(* CoDeSys 2.3.9.41 project: VOS_Vorkuta_ASU_3_osmos_2.pro *)
(* Libraries: PID_Regulators.lib 6.11.19 15:29:27, GermesLib_1_3.lib 17.9.20 11:40:29, Util.lib 18.5.10 15:14:28, STANDARD.LIB 4.10.05 11:14:46, IECSFC.LIB 13.4.06 15:51:28, SYSLIBTIME.LIB 6.11.19 15:29:28, ANALYZATION.LIB 5.10.99 09:05:06 *)

(* PLC configuration (modules and I/O channels)
Fast discrete inputs [I_SIMPLE_INPUT] node 0, in %IB0 out %QB0 {ChannellName = Fast discrete inputs; Filtrationtime = 10000}
  DD1_DI_1 AT %IX0.0 [BitInput] Авария насоса Р03.01/01 {ChannellName = Enter name}
  DD1_DI_2 AT %IX0.1 [BitInput] Авария насоса Р03.01/02 {ChannellName = Enter name}
  DD1_DI_3 AT %IX0.2 [BitInput] эк.манометр PIS03.01/01 после насоса Р03.01/01 {ChannellName = Enter name}
  DD1_DI_4 AT %IX0.3 [BitInput] эк.манометр PIS03.01/02 после насоса Р03.01/02 {ChannellName = Enter name}
Discrete inputs [ID130] node 1, in %IB1 out %QB1 {ChannellName = Discrete inputs; Filtrationtime_GeneralINP = 10; PinCount = 12; Visibility = No}
  AT %IB1.0 [ByteInput] 8 discrete inputs {ChannellName = Enter name}
  AT %IB1.1 [ByteInput] 4 discrete inputs {ChannellName = Enter name}
Fast discrete outputs [OWEN_ID570] node 2, in %IB2 out %QB2 {ChannellName = Fast discrete outputs; SafeValueBool = FALSE; SafeValueBool = FALSE; SafeValueBool = FALSE; SafeValueBool = FALSE; Visibility = No}
  AT %QX2.0 [BitOutput] Fast discrete output 1 {ChannellName = Enter name}
  AT %QX2.1 [BitOutput] Fast discrete output 2 {ChannellName = Enter name}
  AT %QX2.2 [BitOutput] Fast discrete output 3 {ChannellName = Enter name}
  AT %QX2.3 [BitOutput] Fast discrete output 4 {ChannellName = Enter name}
Discrete outputs [ID131] node 3, in %IB3 out %QB3 {ChannellName = Discrete outputs; SafeValueByte = 0; Visibility = No}
  AT %QB3.0 [ByteOutput] 8 discrete outputs {ChannellName = Enter name}
  AT %QB3.1 [ByteOutput] 8 discrete outputs {ChannellName = Enter name}
DD1_AI_1 AT %IR4.0 [FloatInputP] резерв {ChannellName = Fast analog input; AIN_TYPE = 0-20 mA; Peak_Filtr = 200; Flt_Ch = Off; TauRC = 10; MinFV = 0; MaxFV = 20}
DD1_AI_2 AT %IR4.1 [FloatInputP] датчик давления РТ03.01/01 {ChannellName = Fast analog input; AIN_TYPE = 0-20 mA; Peak_Filtr = 200; Flt_Ch = Off; TauRC = 10; MinFV = 0; MaxFV = 20}
DD1_AI_3 AT %IR4.2 [FloatInputP] датчик давления РТ03.02/01 {ChannellName = Fast analog input; AIN_TYPE = 0-20 mA; Peak_Filtr = 200; Flt_Ch = Off; TauRC = 10; MinFV = 0; MaxFV = 20}
DD1_AI_4 AT %IR4.3 [FloatInputP] датчик давления РТ03.03/01 {ChannellName = Fast analog input; AIN_TYPE = 0-20 mA; Peak_Filtr = 200; Flt_Ch = Off; TauRC = 10; MinFV = 0; MaxFV = 20}
DD1_AI_5 AT %IR4.4 [FloatInputP] датчик давления РТ03.04/01 {ChannellName = Fast analog input; AIN_TYPE = 0-20 mA; Peak_Filtr = 200; Flt_Ch = Off; TauRC = 10; MinFV = 0; MaxFV = 20}
DD1_AI_6 AT %IR4.5 [FloatInputP] кондуктомер QIT03.01/01 осн.осмос {ChannellName = Fast analog input; AIN_TYPE = 0-20 mA; Peak_Filtr = 200; Flt_Ch = Off; TauRC = 10; MinFV = 0; MaxFV = 20}
DD1_AI_7 AT %IR4.6 [FloatInputP] расходомер FIT03.02/01 осн.осмос {ChannellName = Fast analog input; AIN_TYPE = 0-20 mA; Peak_Filtr = 200; Flt_Ch = Off; TauRC = 10; MinFV = 0; MaxFV = 20}
DD1_AI_8 AT %IR4.7 [FloatInputP] расходомер FIT03.03/01 осн.осмос {ChannellName = Fast analog input; AIN_TYPE = 0-20 mA; Peak_Filtr = 200; Flt_Ch = Off; TauRC = 10; MinFV = 0; MaxFV = 20}
AT %IW4.8 [WordInput] AI read time (10ms) {ChannellName = Enter name}
Analog outputs [ID126] node 5, in %IB5 out %QB5 {ChannellName = Analog outputs}
  DD1_AO_1 AT %QR5.0 [FloatOutputP] производительность осн.доз.насоса Р03.02/01 {ChannellName = Analog output; AOUT_TYPE = 4-20 mA; SafeValueREAL = 0.0}
  DD1_AO_2 AT %QR5.1 [FloatOutputP] производительность рез.доз.насоса Р03.02/02 {ChannellName = Analog output; AOUT_TYPE = 4-20 mA; SafeValueREAL = 0.0}
  DD1_AO_3 AT %QR5.2 [FloatOutputP] резерв {ChannellName = Analog output; AOUT_TYPE = 4-20 mA; SafeValueREAL = 0.0}
  DD1_AO_4 AT %QR5.3 [FloatOutputP] резерв {ChannellName = Analog output; AOUT_TYPE = 4-20 mA; SafeValueREAL = 0.0}
Special input [ID103] node 6, in %IB6 out %QB6 {ChannellName = Special input}
  AT %IX6.0 [BitInput] Special input {ChannellName = Enter name}
Special output [ID104] node 7, in %IB7 out %QB7 {ChannellName = Special output}
  AT %QX7.0 [BitOutput] Special output {ChannellName = Enter name}
AT %QD8.0 [DWordOutput] Last address {ChannellName = Enter name}
AT %QW8.1 [WordOutput] Last error {ChannellName = Enter name}
RS-485-1 [COM1_USART] node 0, in %IB8.0 out %QB8.0 {ChannellName = RS-485-1; CommunicationSpeed = 9600; Parity = NO PARITY CHECK; BitLength = 8 bits; StopLength = One stop bit; InterfaceType = RS485; FrameOriented = RTU; Timeout = 5; Visibility = No}
AT %QB8.1.0 [ComChannel] Command (0xff - Start) {ChannellName = Enter name}
Real input module [ID2007] node 0, in %IB8.1.0 out %QB8.1.0 {ChannellName = float input module; ModbusAddress = 512; Command_read_regs = Read holding Registers  (0x03); Visibility = No}
  PT030102rawValue AT %QD8.1.0.0 [FloatOutput] {ChannellName = Enter name}
Real input module [ID2007] node 1, in %IB8.1.1 out %QB8.1.1 {ChannellName = float input module; ModbusAddress = 514; Command_read_regs = Read holding Registers  (0x03); Visibility = No}
  PT030202rawValue AT %QD8.1.1.0 [FloatOutput] {ChannellName = Enter name}
  PT030302rawValue AT %QD8.1.2.0 [FloatOutput] {ChannellName = Enter name}
Real input module [ID2007] node 3, in %IB8.1.3 out %QB8.1.3 {ChannellName = float input module; ModbusAddress = 518; Command_read_regs = Read holding Registers  (0x03); Visibility = No}
  PT030402rawValue AT %QD8.1.3.0 [FloatOutput] {ChannellName = Enter name}
Real input module [ID2007] node 4, in %IB8.1.4 out %QB8.1.4 {ChannellName = float input module; ModbusAddress = 520; Command_read_regs = Read holding Registers  (0x03); Visibility = No}
  QIT030102rawValue AT %QD8.1.4.0 [FloatOutput] {ChannellName = Enter name}
Real input module [ID2007] node 5, in %IB8.1.5 out %QB8.1.5 {ChannellName = float input module; ModbusAddress = 522; Command_read_regs = Read holding Registers  (0x03); Visibility = No}
  FIT030202rawValue AT %QD8.1.5.0 [FloatOutput] {ChannellName = Enter name}
Real input module [ID2007] node 6, in %IB8.1.6 out %QB8.1.6 {ChannellName = float input module; ModbusAddress = 524; Command_read_regs = Read holding Registers  (0x03); Visibility = No}
  FIT030302rawValue AT %QD8.1.6.0 [FloatOutput] {ChannellName = Enter name}
Real input module [ID2007] node 7, in %IB8.1.7 out %QB8.1.7 {ChannellName = float input module; ModbusAddress = 526; Command_read_regs = Read holding Registers  (0x03); Visibility = No}
  FIT030101rawValue AT %QD8.1.7.0 [FloatOutput] {ChannellName = Enter name}
Register input module [ID2003] node 8, in %IB8.1.8 out %QB8.1.8 {ChannellName = Register input module; ModbusAddress = 529; Command_read_regs = Read input registers  (0x04); Visibility = No}
  DI_bit_mask_DD2 AT %QW8.1.8.0 [WordOutput] {ChannellName = Enter name}
Register input module [ID2003] node 9, in %IB8.1.9 out %QB8.1.9 {ChannellName = Register input module; ModbusAddress = 532; Command_read_regs = Read input registers  (0x04); Visibility = No}
  stat_word_P030601_PLC AT %QW8.1.9.0 [WordOutput] {ChannellName = Enter name}
  stat_word_P030602_PLC AT %QW8.1.10.0 [WordOutput] {ChannellName = Enter name}
Universal Modbus device [ID2000] node 2, in %IB8.2 out %QB8.2 {ChannellName = Universal Modbus device; ModuleIP = 10:0:0:223; ServiceTimeout = 150; TCPport = 502; NetMode = Serial; ModuleSlaveAddress = 1; RequestType = By value change; PeriodOfService = 100; Visibility = No; RepeatCounter = 0; ByteSequence = Native}
  AT %QB8.2.0 [ComChannel] Command (0xff - Start) {ChannellName = Enter name}
  Register output module [ID2004] node 0, in %IB8.2.0 out %QB8.2.0 {ChannellName = Register; ModbusAddress = 528; Command_write_one_reg = Write multiple registers(0x10); Visibility = No}
    DO_bit_mask_DD2 AT %QW8.2.0.0 [WordOutput] {ChannellName = Enter name}
  Register output module [ID2004] node 1, in %IB8.2.1 out %QB8.2.1 {ChannellName = Register; ModbusAddress = 530; Command_write_one_reg = Write multiple registers(0x10); Visibility = No}
    com_word_P030601_PLC AT %QW8.2.1.0 [WordOutput] {ChannellName = Enter name}
  Register output module [ID2004] node 2, in %IB8.2.2 out %QB8.2.2 {ChannellName = Register; ModbusAddress = 531; Command_write_one_reg = Write multiple registers(0x10); Visibility = No}
    set_freq_P030601_PLC AT %QW8.2.2.0 [WordOutput] {ChannellName = Enter name}
  Register output module [ID2004] node 3, in %IB8.2.3 out %QB8.2.3 {ChannellName = Register; ModbusAddress = 533; Command_write_one_reg = Write multiple registers(0x10); Visibility = No}
    com_word_P030602_PLC AT %QW8.2.3.0 [WordOutput] {ChannellName = Enter name}
    set_freq_P030602_PLC AT %QW8.2.4.0 [WordOutput] {ChannellName = Enter name}
RS-232 [COM2_USART] node 0, in %IB9.0.0 out %QB9.0.0 {ChannellName = RS-232; CommunicationSpeed = 115200; Parity = NO PARITY CHECK; BitLength = 8 bits; StopLength = One stop bit; InterfaceType = RS232; FrameOriented = RTU; Timeout = 0; Visibility = No}
*)

(* POU PLC_PRG, CFC *)
PROGRAM PLC_PRG
VAR
	boolStub: BOOL; (*Заглушка bool*)
	realStub: REAL; (*Заглушка real*)
	P0301: RichTwoPumpManager;		(*управление насосами Р03.01 на входе в осмос*)
	resetAlarms: BOOL;		(*Сброс аварий в осмос 2 (МЕ03)*)
	delayCheckIfP030101works: TON;		(*задержка на разгон насоса Р03.01/01*)
	delayCheckIfP030102works: TON;		(*задержка на разгон насоса Р03.01/02*)
	statWordP0301: WORD;		(*статусы состояния насосов Р03.01*)
	lowLevelV0207: BOOL;		(*низкий уровень в емкости V02.07, сигнал из АСУ-2 осмос-1*)
	highLevelV0601: BOOL;		(*высокий уровень в емкости V06.01 сигнал из АСУ-1 общий.*)
	highLevelV0401: BOOL;		(*высокий уровень в емкости V04.01, сигнал из МЕ04, от БМТ.*)
	toNextStarnP030101timer: WORD;		(*Обратный отсчет до возможности повторного пуска насоса Р03.01/01*)
	toNextStarnP030102timer: WORD;		(*обратный отсчет до возможности повторного пуска насоса Р03.01/02*)
	flowFIT0301: REAL;		(*Показания расходомера FIT03.01/01 на входе в осмос 2.
			Для управления производительностью НД Р03.02 (1 и 2).*)
	P0302: RichTwoPumpManager;		(*блок управления доз.насосами Р03.02/01 и Р03.02/02.*)
	statWordP0302: WORD;		(*Статусы состояния доз.насосов Р03.02 на входе осмос 2.*)
	P0302dos: DosingPumpProportional;		(*блок управления промзводительностью доз.насосов Р03.02.*)
	setMaxPumpDosingValueP0302: REAL;		(*задание максимальной производительности доз.насоса, в мл/мин*)
	setKoeffProportionalityP0302: REAL;		(*Задание мл на кубометр (коэф.пропорциональности между расходом и дозированием)*)
	dosingErrorP0302: BOOL;		(*Ошибка производительности дозирования (неверно заданы значения производительности насоса,
производительность доз.насоса не соответствует расходу.*)
	initializer: R_TRIG;		(*триггер дающий импульс при включении программы.*)
	alarmP0302: BOOL;		(*авария обоих доз.насосов Р03..02 на входе в осмос*)
	osmosTotalAlarm: BOOL;		(*авария обоих осмосов*)
	controlAIpt030101: ControlAI;
	PT030101realValue: REAL;		(*Показания датчика РТ03.01/01, МПа (Бар)*)
	PT030101alarm: BOOL;		(*авария датчика РТ03.01/01*)
	controlAIpt030201: ControlAI;
	PT030201realValue: REAL;
	PT030201alarm: BOOL;
	controlAIpt030301: ControlAI;
	PT030301realValue: REAL;
	PT030301alarm: BOOL;
	controlAIpt030401: ControlAI;
	PT030401realValue: REAL;
	PT030401alarm: BOOL;
	controlAIqit030101: ControlAI;
	QIT030101realValue: REAL;
	QIT030101alarm: BOOL;
	controlAIfit030201: ControlAI;
	FIT030201realValue: REAL;
	FIT030201alarm: BOOL;
	controlAIfit030301: ControlAI;
	FIT030301realValue: REAL;
	FIT030301alarm: BOOL;
	osmos2sensorsAlarm: BOOL;		(*Авария датчиков осмос 2.
			в DD2 (ПР102) есть авария одного из датчиков.*)
	osmosManager: RichTwoPumpManager;
	toNextStarnOsmos1timer: WORD;
	toNextStarnOsmos2timer: WORD;
	minutesOfWorkOsmos2: WORD;
	secondsOfWorkOsmos2: WORD;
	osmos1SensorAlarm: BOOL;		(*Авария оборудования основного осмоса.*)
	osmos1EquipmentAlarm: BOOL;		(*Авария оборудования основного осмоса.*)
	osmos2EquipmentAlarm: BOOL;		(*авария оборудования резервного осмоса*)
	tofValve12: TOF;
	tonValve14: TON;
	tofValve14: TOF;
	tonValve18: TON;
	startP0302: BOOL;		(*сигнал на запуск насосов-дозаторов Р03.02*)
	tonPT030101: TON;
	lowPT030101_P030101: BOOL;		(*давление на РТ030101 не достигло значения для старта при
			активном насосе Р03.01/01*)
	lowPT030101_P030102: BOOL;		(*давление на РТ030101 не достигло значения для старта при
			активном насосе Р03.01/02*)
	tonSwitchValve1413: TON;
	valve1413switcher: IfBOOL;
	delayToSwitchValve14to13: TOF;
	F_P030601: PID;		(*PID регулятор по расходу Р03.06/01*)
	P_P030601: PID;		(*PID регулятор по давлению Р03.06/01*)
	Yout_F_P030601: REAL;		(*задание ПИД по расходу для Р030601*)
	Yout_P_P030601: REAL;		(*выход регулировки по давлению Р03.06/01, 0...100*)
	Yout_Total_P030601: REAL;		(*итоговый управляющий сигнал производительность Р03.06/01*)
	Yout_F_P030602: REAL;		(*задание ПИД по расходу для Р030602*)
	Yout_P_P030602: REAL;		(*выход регулировки по давлению Р03.06/02, 0...100*)
	Yout_Total_P030602: REAL;		(*итоговый управляющий сигнал производительность Р03.06/02*)
	P030601alarm: BOOL;		(*авария насоса Р03.06/01*)
	P030602alarm: BOOL;		(*авария насоса Р03.06/02*)
	P030601start: BOOL;		(*сигнал на запуск насоса Р03.06/01*)
	P030602start: BOOL;		(*сигнал на запуск насоса Р03.06/02*)
	osmos1AlarmPT030301: BOOL;		(*авария основного осмоса по макс давлению датчика РТ03.03/01*)
	osmos1AlarmPT030401: BOOL;		(*авария основного осмоса по макс давлению датчика РТ03.04/01*)
	osmos2AlarmPT030302: BOOL;		(*авария основного осмоса по макс давлению датчика РТ03.03/02*)
	osmos2AlarmPT030402: BOOL;		(*авария основного осмоса по макс давлению датчика РТ03.04/02*)
	tofValve18: TOF;
	HoldingToEndProcValve: TOF;
	tonValve17: TON;
	tonValve18rez: TON;
	tofValve18rez: TOF;
	tofValve17: TOF;
	tofValve15: TOF;
	lowPT030102_P030101: BOOL;		(*авария насоса Р03.01/01 по низкому давлению РТ03.01/02*)
	lowPT030102_P030102: BOOL;		(*авария насоса Р03.01/02 по низкому давлению РТ03.01/02*)
	PT030102realValue: REAL;		(*давление РТ03.01/02 из DD2*)
	tonSwitchValve1716: TON;
	HoldingToEndProcValveRez: TOF;
	tonPT030102: TON;
	valve1716switcher: IfBOOL;
	delayToSwitchValve17to16: TOF;
	PT030202realValue: REAL;
	PT030302realValue: REAL;
	PT030402realValue: REAL;
	FIT030302realValue: REAL;
	F_P030602: PID;
	P_P030602: PID;
	statWordOsmos: WORD;		(*статус состояни осмосов*)
	FIT030202realValue: REAL;
	QIT030102realValue: REAL;
	freqP030601: LIN_TRAFO;
	freqP030602: LIN_TRAFO;
	pt030102:ControlAI;
	pt030202: ControlAI;
	pt030302: ControlAI;
	pt030402: ControlAI;
	fit0301: ControlAI;
	fit030202: ControlAI;
	qit030102: ControlAI;
	fit030302:ControlAI;
	PT030102alarm: BOOL;		(*авария датчика*)
	PT030202alarm: BOOL;
	PT030302alarm: BOOL;
	PT030402alarm: BOOL;
	FIT0301alarm: BOOL;
	FIT030202alarm: BOOL;
	FIT030302alarm: BOOL;
	QIT030102alarm: BOOL;

	testReal: REAL;
	testReal1: REAL;
	testReal2: REAL;
	testBool1: BOOL;
	testBool2: BOOL;
	testBlink: BLINK;
END_VAR
VAR RETAIN
	counterP030101: DWORD;		(*счетчик включений насоса Р03.01/01*)
	counterP030102: DWORD;		(*счетчик включений насоса Р03.01/02*)
	daysOfWorkP030101: WORD;		(*количество дней работы насоса Р03.01/01*)
	daysOfWorkP030102: WORD;		(*количество дней работы насоса Р03.01/02*)
	hoursOfWorkP030101: WORD;		(*количество часов работы насоса Р03.01/01*)
	hoursOfWorkP030102: WORD;		(*количество часов работы насоса Р03.01/02*)
	minutesOfWorkP030101: WORD;		(*количество минут работы Р03.01/01*)
	minutesOfWorkP030102: WORD;		(*количество минут работы насоса Р03.01/02*)
	secondsOfWorkP030101: WORD;		(*количество секунд работы насоса Р03.01/01*)
	secondsOfWorkP030102: WORD;		(*количество секунд работы насоса Р03.01/02*)
	counterP030201: DWORD;
	counterP030202: DWORD;
	daysOfWorkP030201: WORD;
	daysOfWorkP030202: WORD;
	hoursOfWorkP030201: WORD;
	hoursOfWorkP030202: WORD;
	minutesOfWorkP030201: WORD;
	minutesOfWorkP030202: WORD;
	secondsOfWorkP030201: WORD;
	secondsOfWorkP030202: WORD;
	toNextStarnP030201timer: WORD;
	toNextStarnP030202timer: WORD;
	setWordP0301: WORD;		(*конфигурация работы Р0301*)
	setWordP0302: WORD;		(*Конфигурация работы доз.насосов Р03.01*)
	PT030101maxValue: REAL;		(*Максимальное значение показаний датчика РТ03.01/01
			(при 20мА)*)
	PT030201maxValue: REAL;
	PT030301maxValue: REAL;
	PT030401maxValue: REAL;
	QIT030101maxValue: REAL;
	FIT030201maxValue: REAL;
	FIT030301maxValue: REAL;

	PT030102maxValue: REAL;
	PT030202maxValue: REAL;
	PT030302maxValue: REAL;
	PT030402maxValue: REAL;
	FIT0301maxValue: REAL;
	FIT030202maxValue: REAL;
	FIT030302maxValue: REAL;
	QIT030102maxValue: REAL;

	counterOsmos1: DWORD;
	counterOsmos2: DWORD;
	daysOfWorkOsmos1: WORD;
	hoursOfWorkOsmos1: WORD;
	minutesOfWorkOsmos1: WORD;
	secondsOfWorkOsmos1: WORD;
	daysOfWorkOsmos2: WORD;
	hoursOfWorkOsmos2: WORD;
	PT0301startValue: REAL;		(*Давление РТ0301 для запуска насоса*)
	FIT0303setValue: REAL;		(*Задание расхода для осмоса*)
	PT0303setValue: REAL;		(*Задание максимального давления на РТ03.03*)
	PT0303setMaxValue: REAL;		(*Задание максимального давления на РТ03.03*)
	KP_F_P030601: REAL := 1;
	I_F_P030601: REAL := 10;
	D_F_P030601: REAL := 1;
	KP_P_P030601: REAL := 1;
	I_P_P030601: REAL := 10;
	D_P_P030601: REAL := 1;
	KP_F_P030602: REAL := 1;
	I_F_P030602: REAL := 10;
	D_F_P030602: REAL := 1;
	KP_P_P030602: REAL := 1;
	I_P_P030602: REAL := 10;
	D_P_P030602: REAL := 1;
	PT0302setMaxValue: REAL;
	PT0304setMaxValue: REAL;
	DELAY_TO_CLOSE_VALVE: TIME;		(*задержка до начала закрытия клапанов после выключения насосов*)
	DELAY_TO_SWITCH_VALVE: TIME;		(*время задержки до переключения клапанов после запуска насоса Р0306*)
	DELAY_TO_CHECK_PT0301: TIME;
	DELAY_TO_OFF_VALVE: TIME;
	DELAY_REPEATED_START_SEC: WORD;		(*время задержки повторного пуска насосов, сек, защита от частых пусков*)
	CHECKING_DELAY_TIME: TIME;		(*время задержки начала контроля параметра (например, задержка
			контроля эк.манометра после насоса, время на разгон).*)
	setWordOsmos: WORD;		(*Конфигурация режимов работы осмосов*)
END_VAR
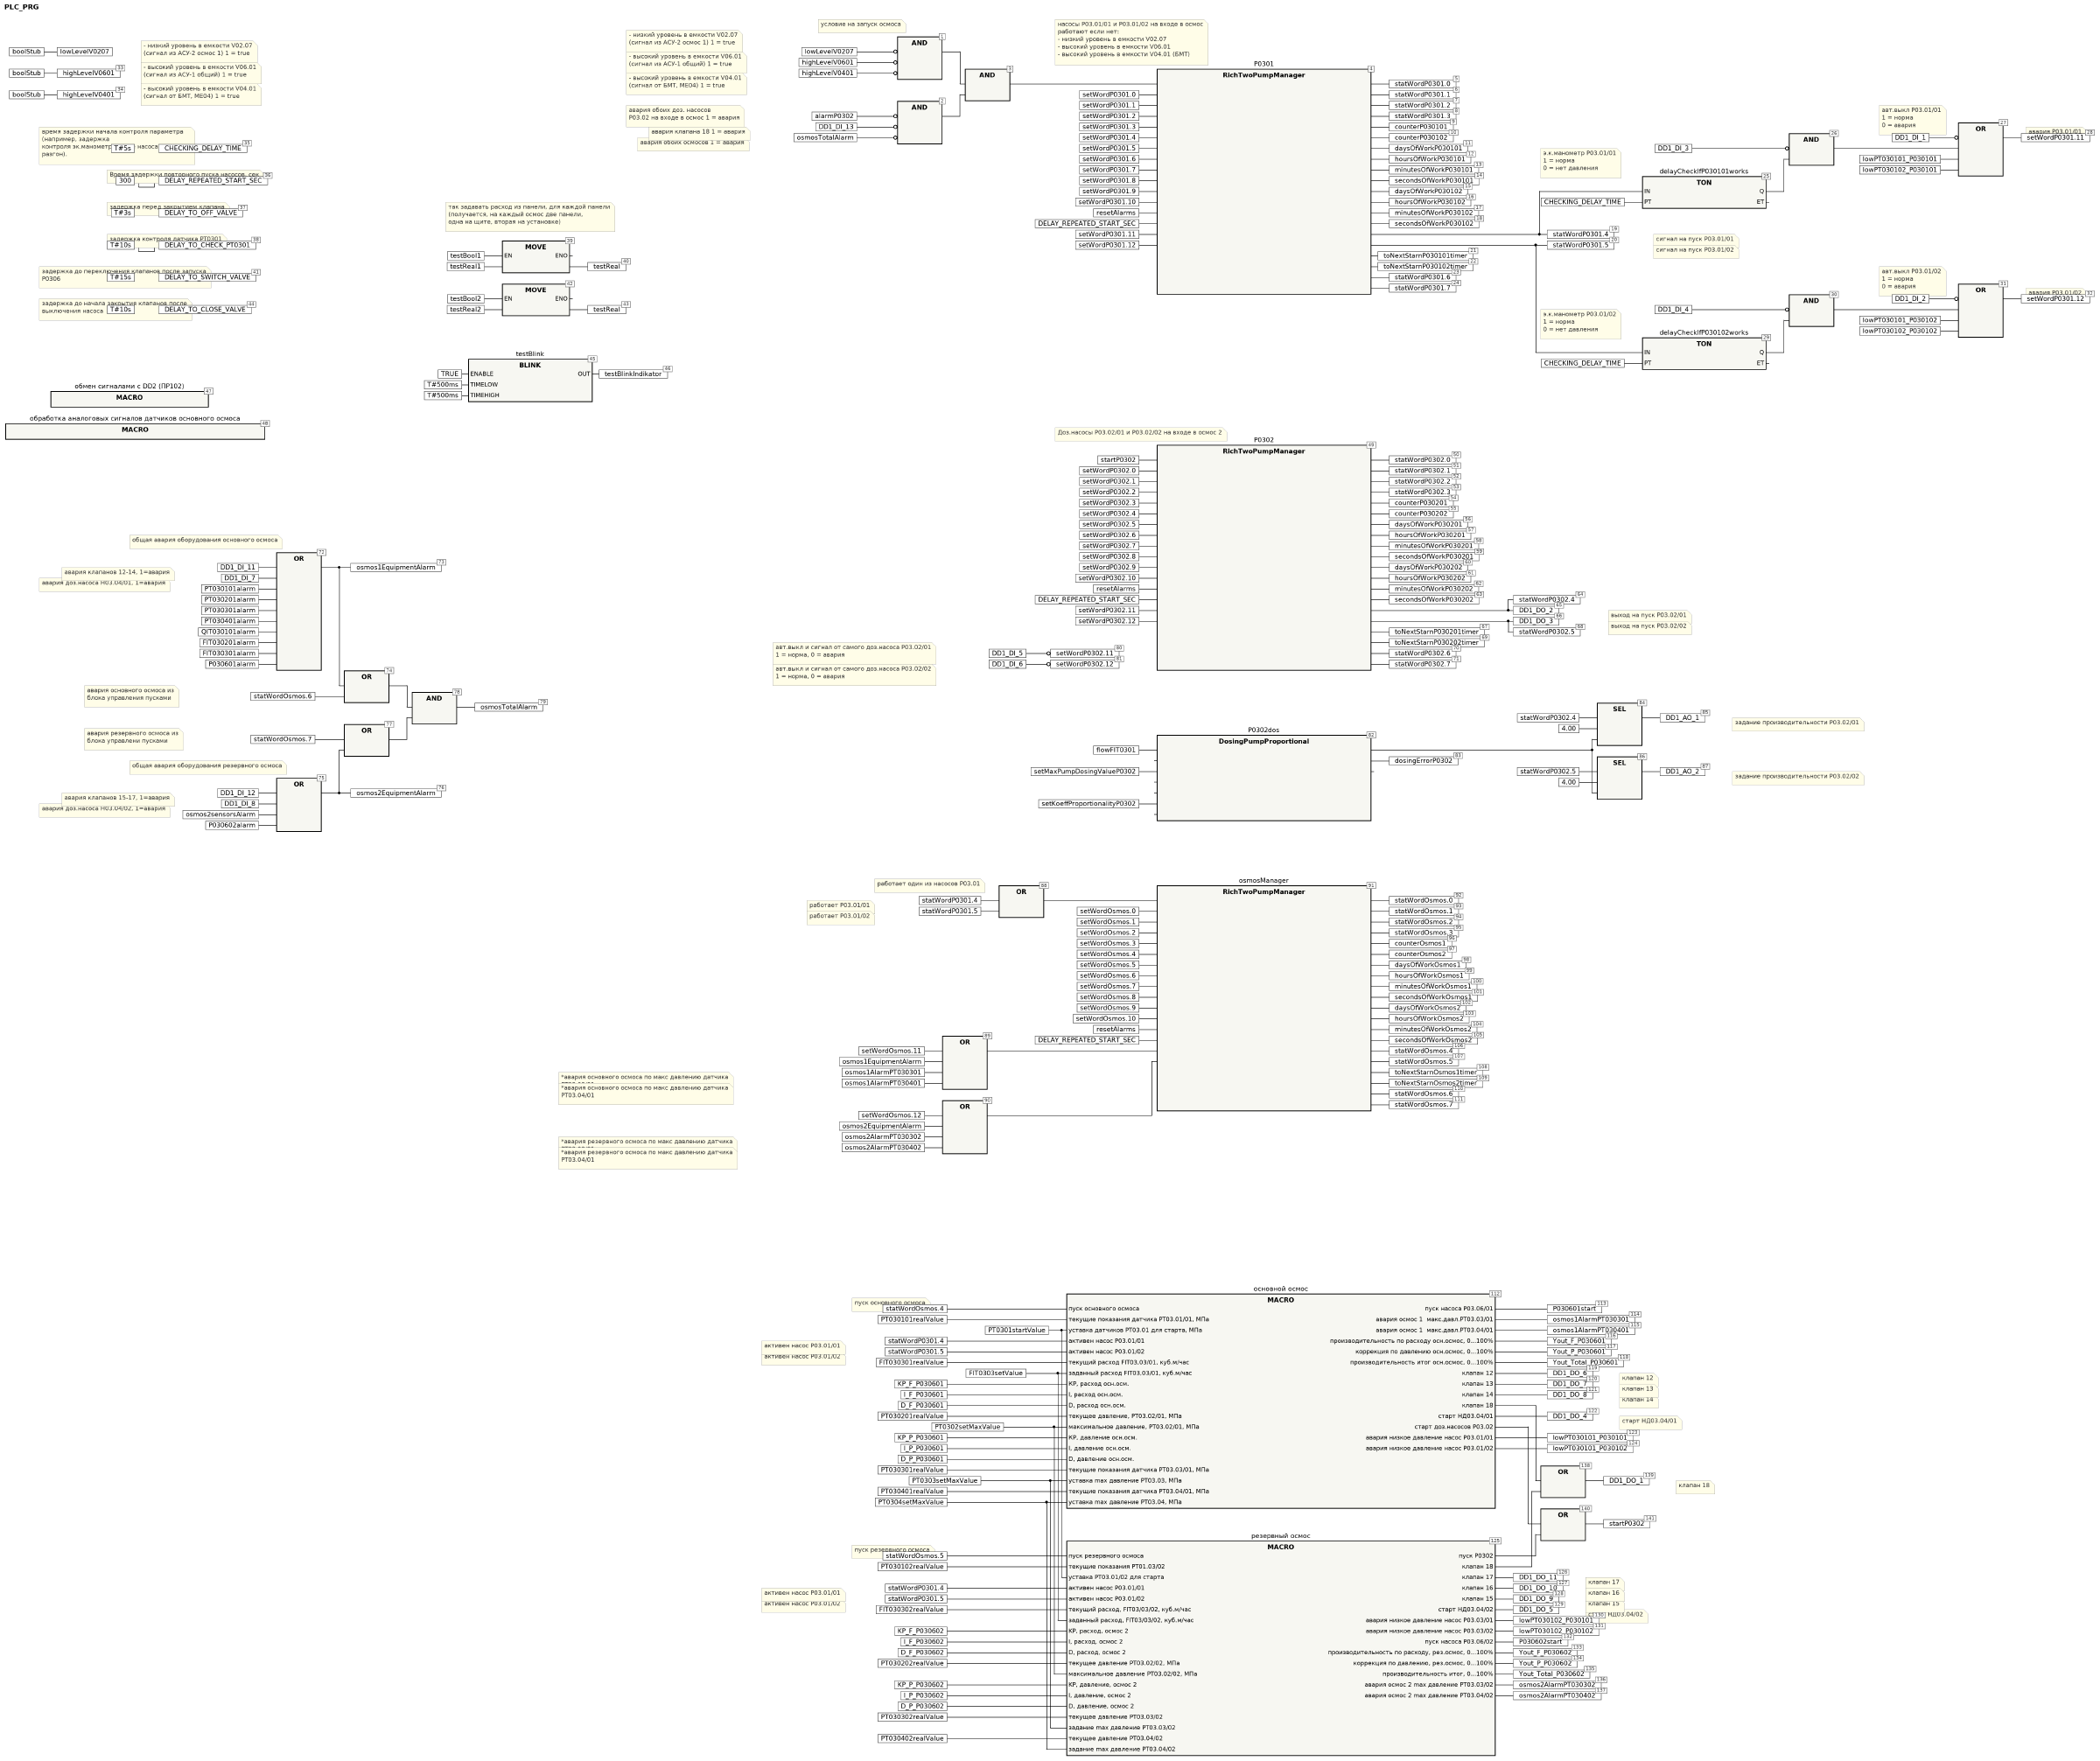
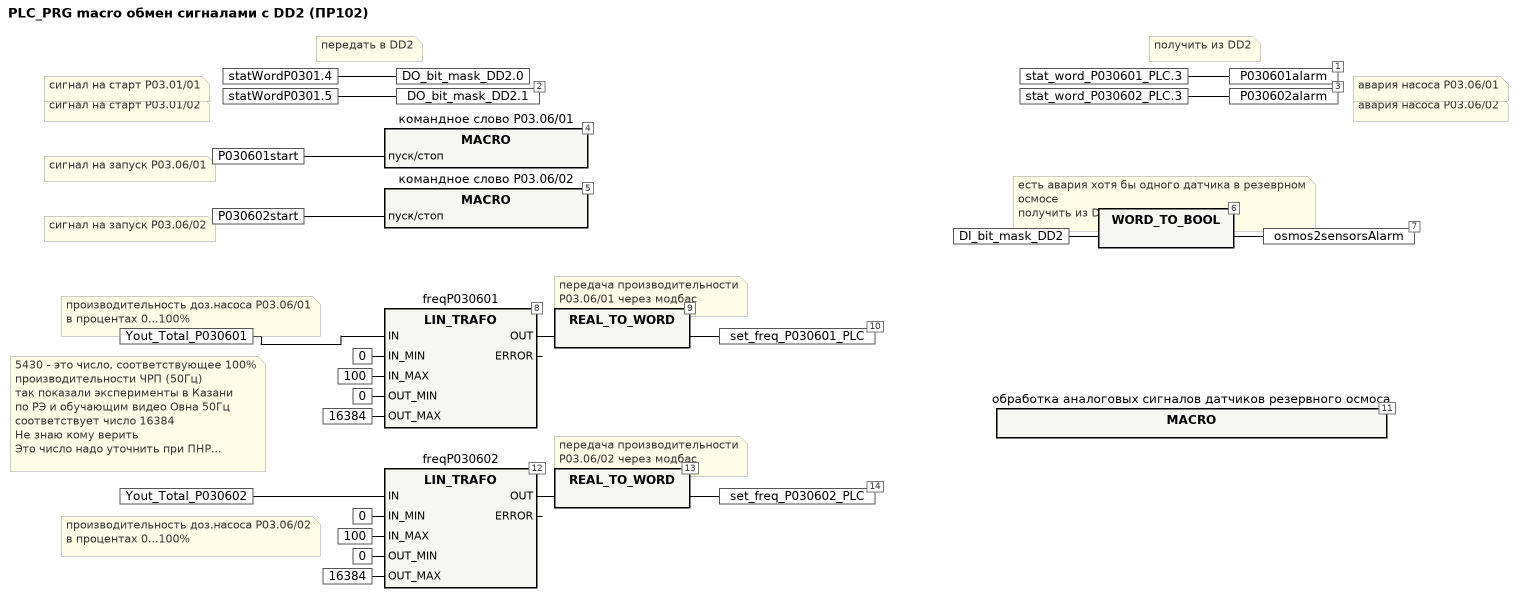
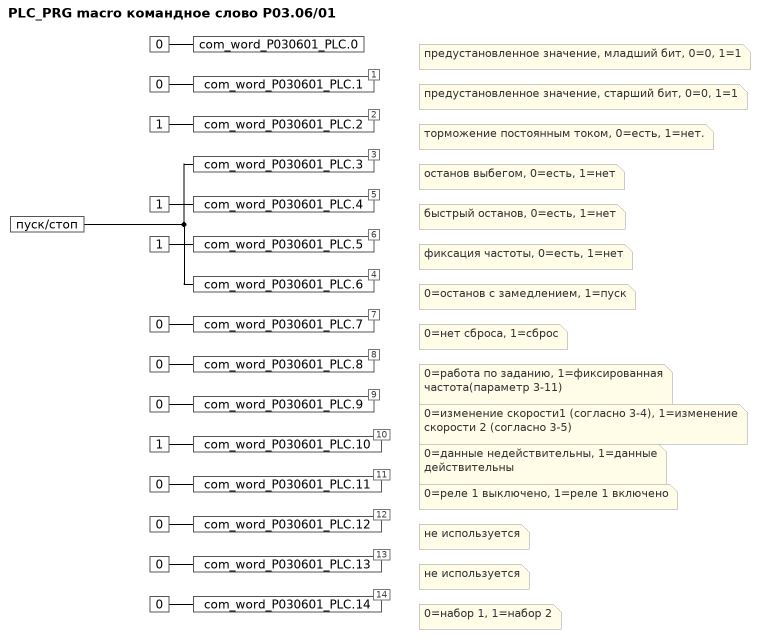
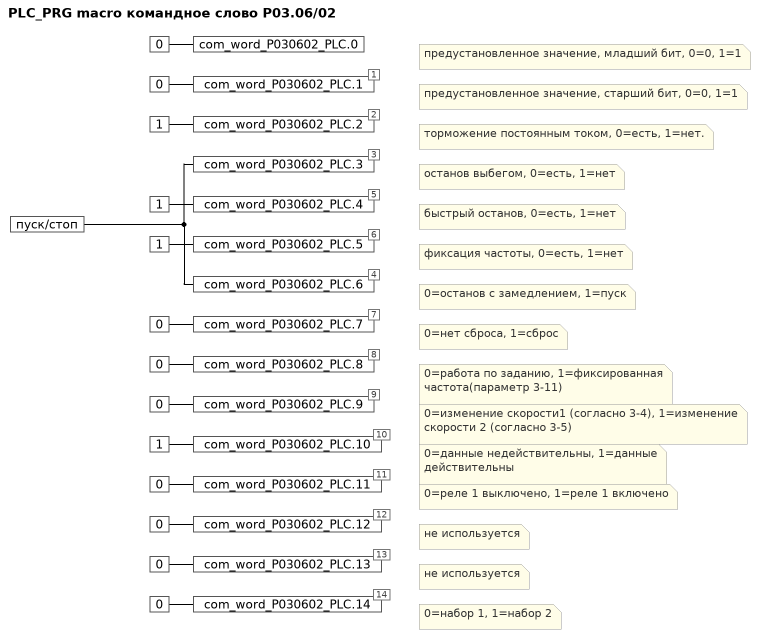
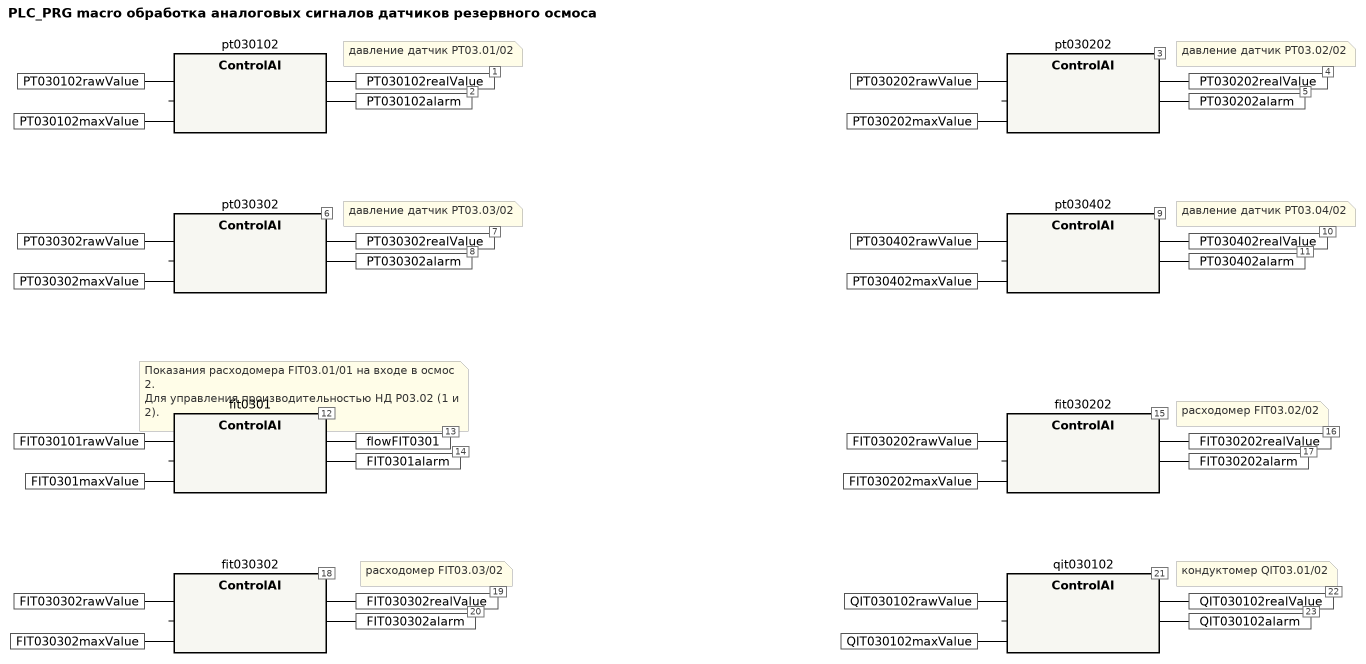
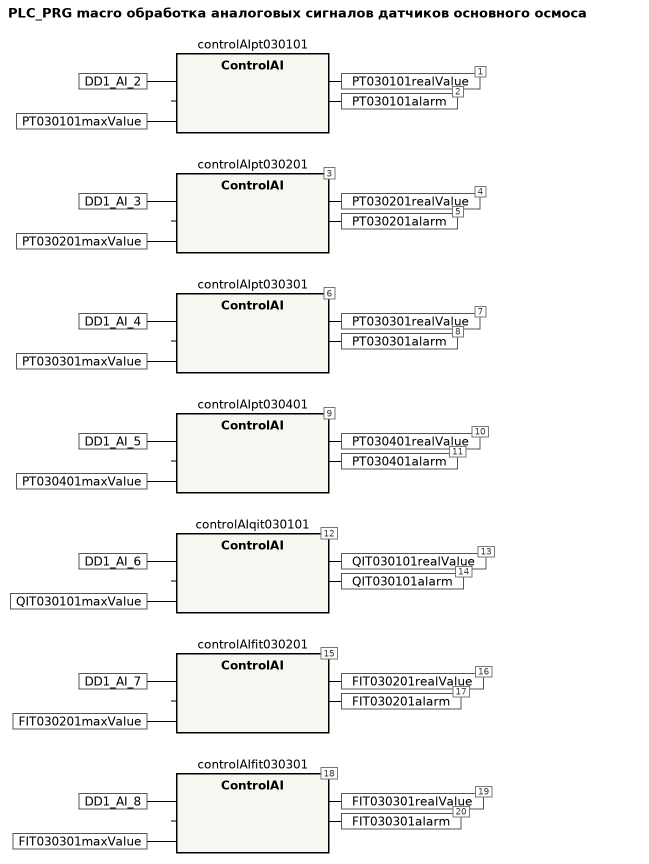
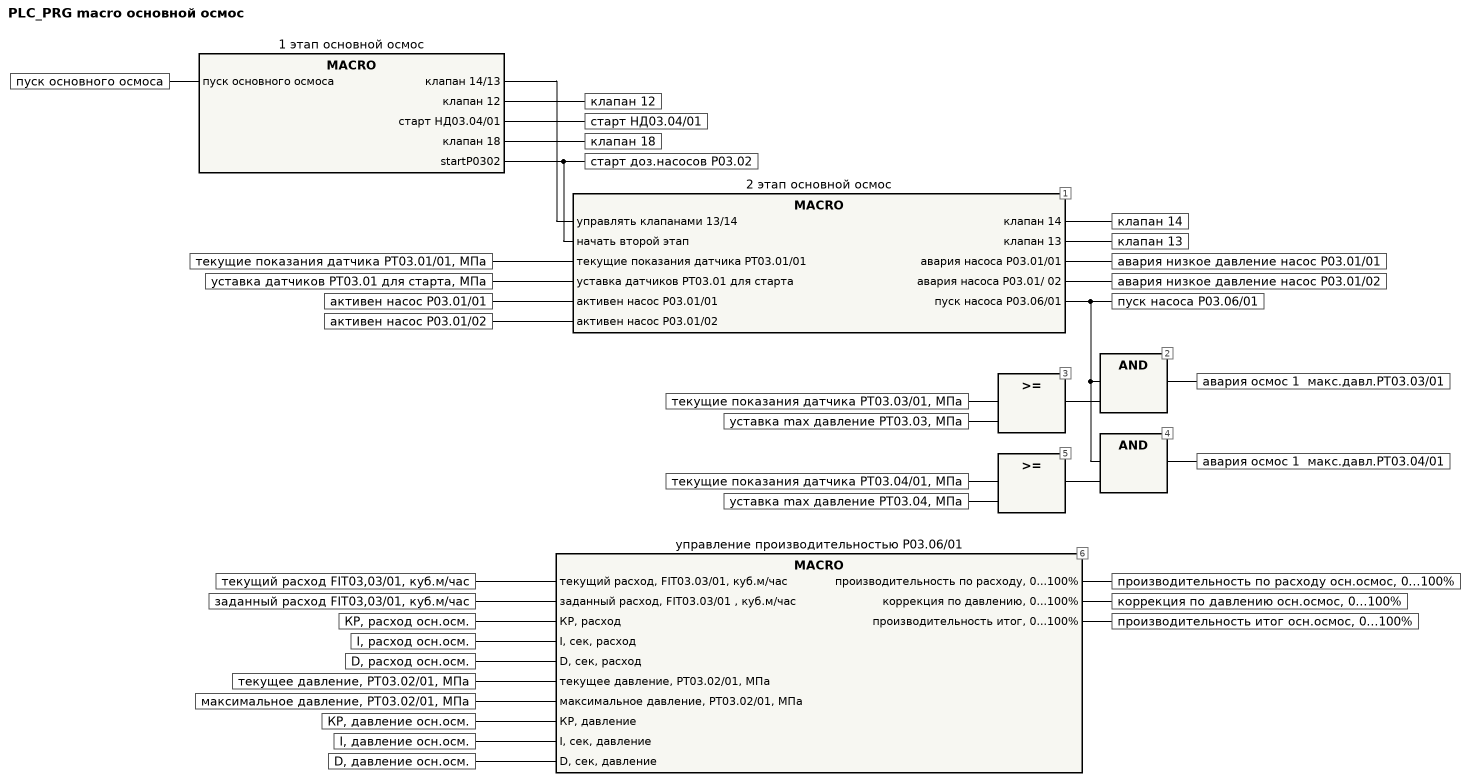
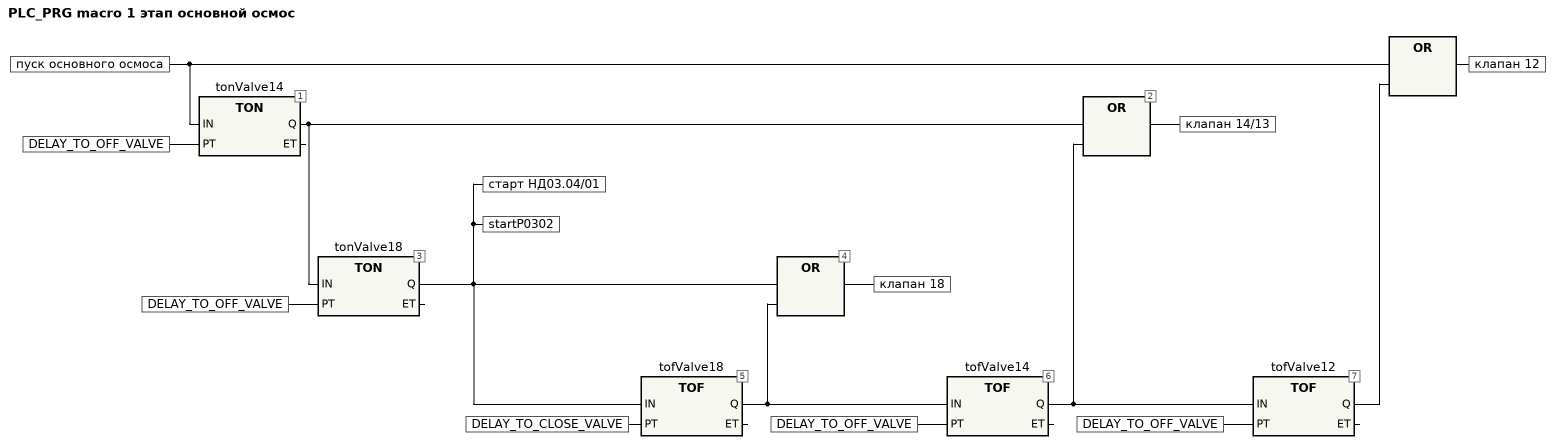
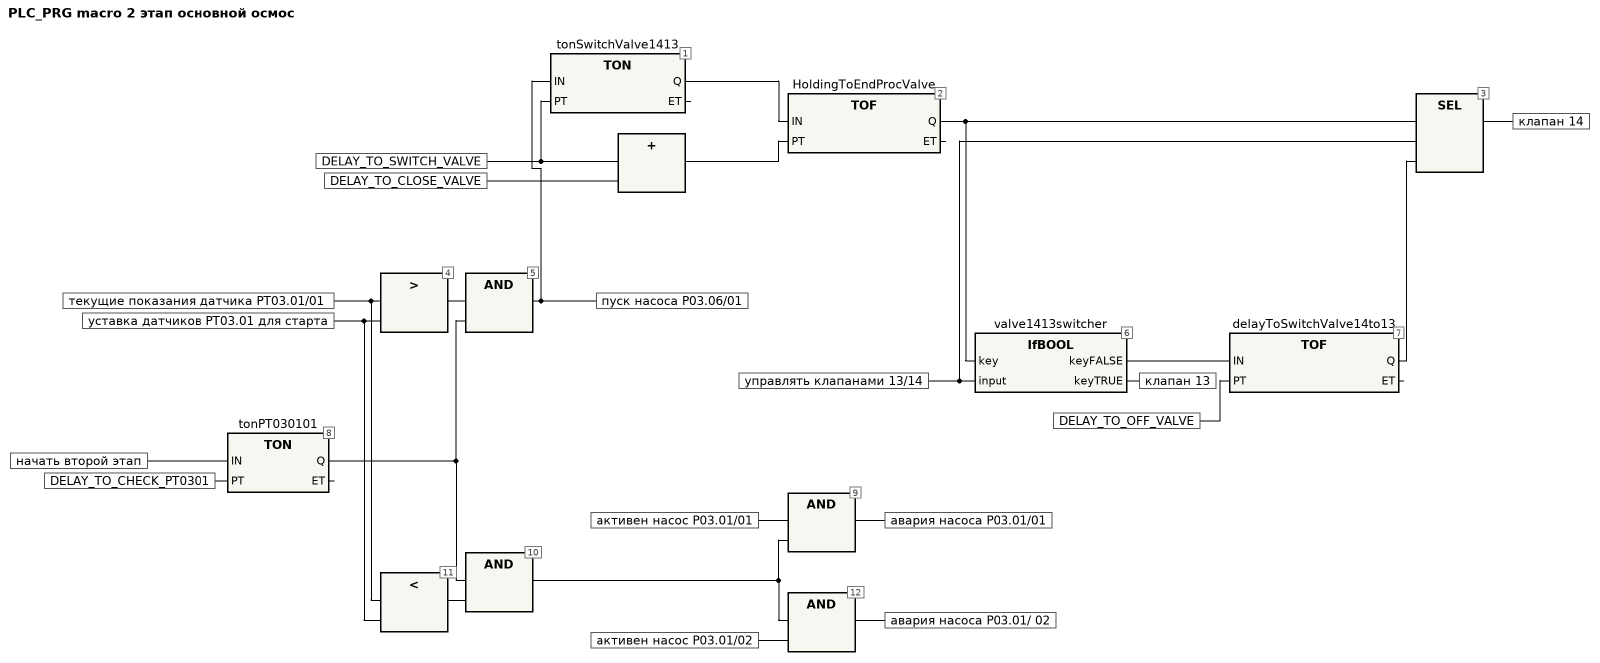
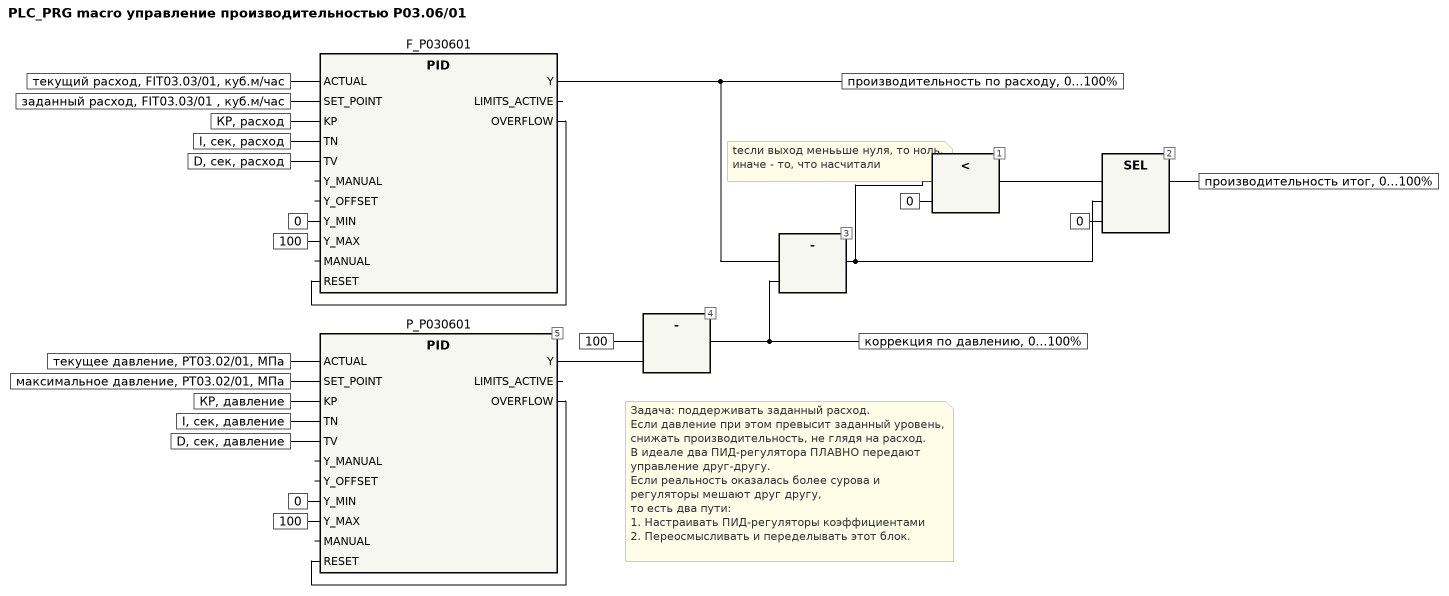
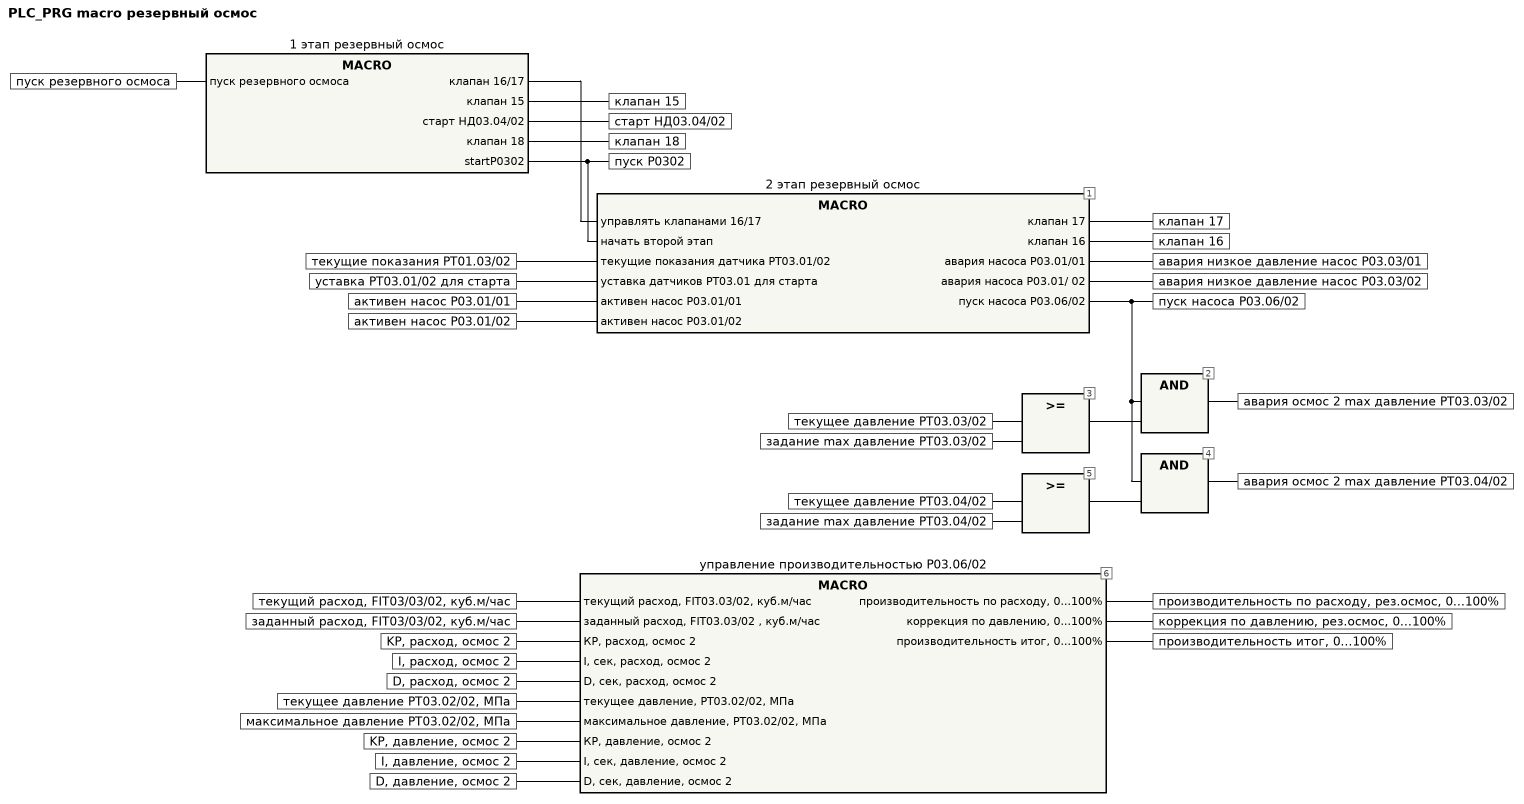
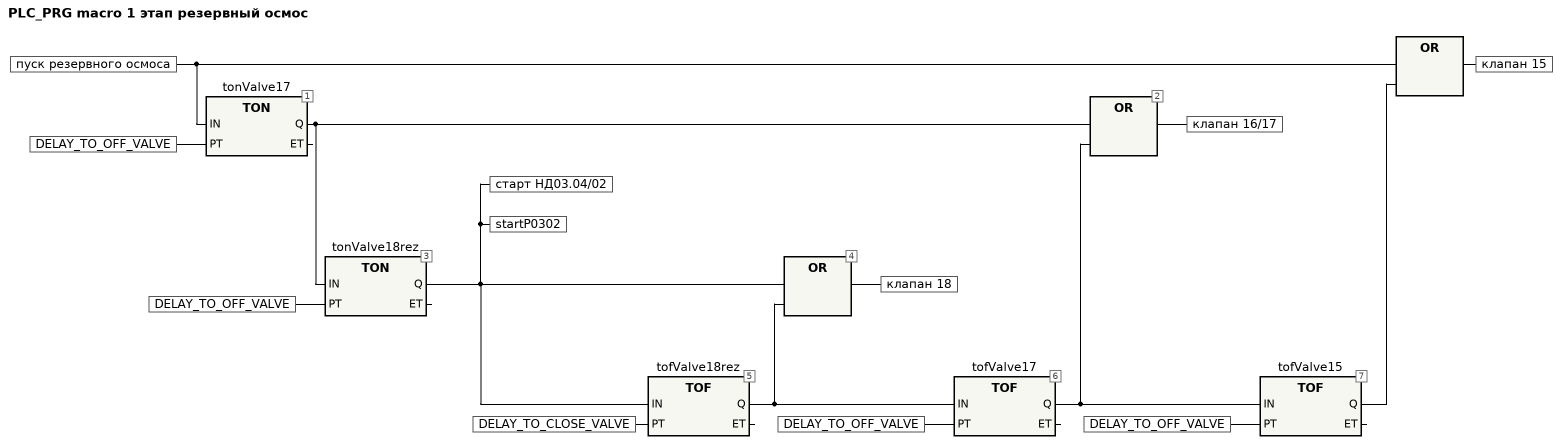
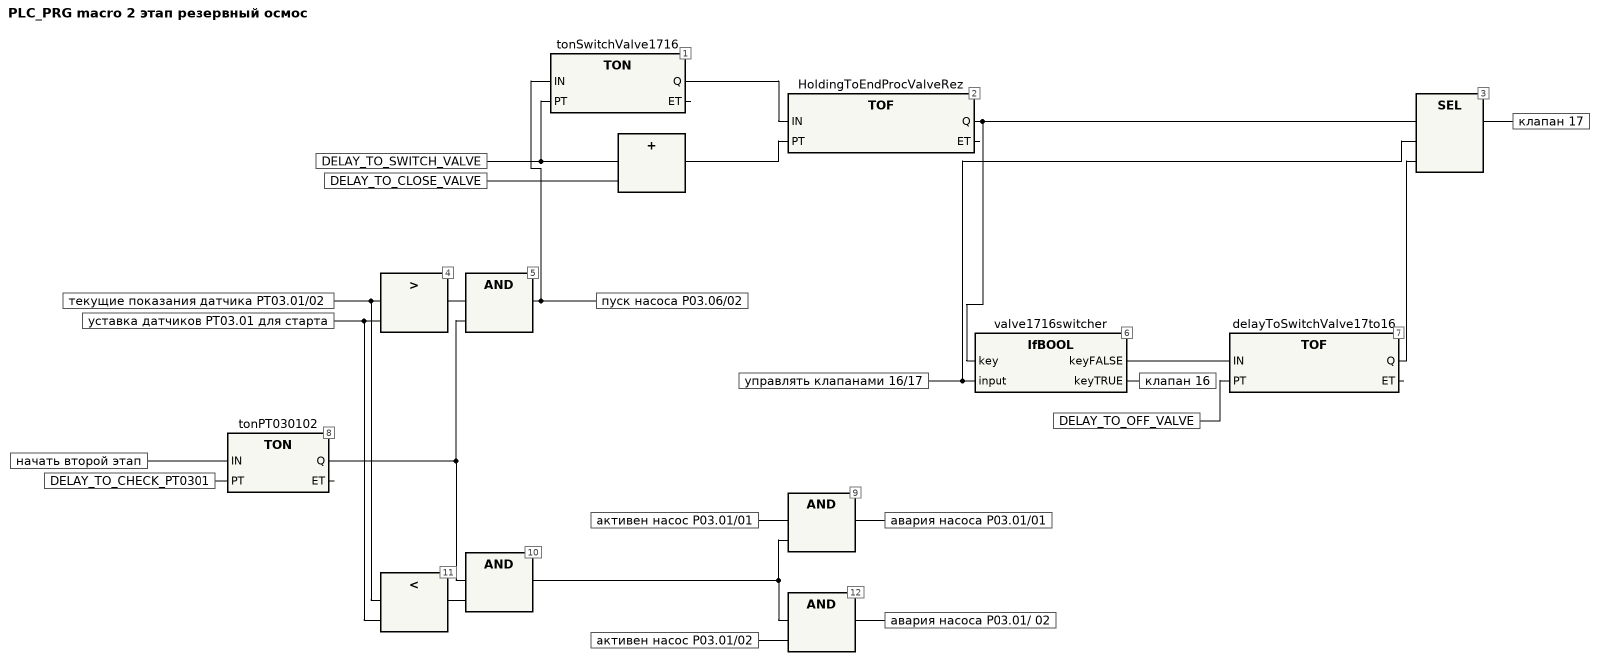
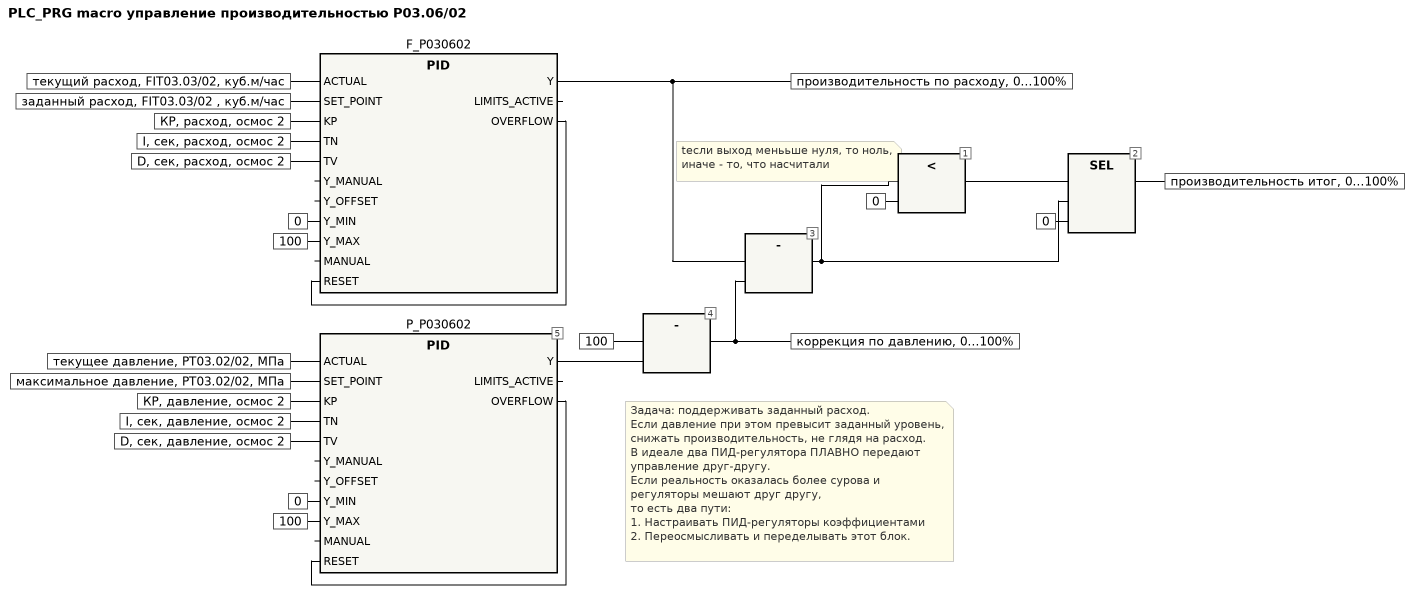
_CFC_ (* Continuous Function Chart, elements in execution order *)
(* так задавать расход из панели, для каждой панели / (получается, на каждый осмос две панели, / одна на щите, вторая на установке) *)
(* активен насос Р03.01/02 *)
(* активен насос Р03.01/01 *)
(* старт НД03.04/01 *)
(* задержка до переключения клапанов после запуска Р0306 *)
(* задержка перед закрытием клапана *)
(* работает Р03.01/01 *)
(* работает Р03.01/02 *)
(* работает один из насосов Р03.01 *)
(* авария доз.насоса Н03.04/02, 1=авария *)
(* общая авария оборудования резервного осмоса *)
(* авария клапанов 15-17, 1=авария *)
(* общая авария оборудования основного осмоса *)
(* авария доз.насоса Н03.04/01, 1=авария *)
(* авария клапанов 12-14, 1=авария *)
(* условие на запуск осмоса *)
(* авария обоих осмосов 1 = авария *)
(* авария клапана 18 1 = авария *)
(* авария обоих доз. насосов / Р03.02 на входе в осмос 1 = авария *)
(* насосы Р03.01/01 и Р03.01/02 на входе в осмос / работают если нет: / - низкий уровень в емкости V02.07 / - высокий уровень в емкости V06.01 / - высокий уровень в емкости V04.01 (БМТ) *)
(* - низкий уровень в емкости V02.07 / (сигнал из АСУ-2 осмос 1) 1 = true *)
(* - высокий уровень в емкости V06.01 / (сигнал из АСУ-1 общий) 1 = true *)
(* - высокий уровень в емкости V04.01 / (сигнал от БМТ, МЕ04) 1 = true *)
(* авария Р03.01/01 *)
(* авт.выкл Р03.01/01 / 1 = норма / 0 = авария *)
(* сигнал на пуск Р03.01/01 *)
(* авт.выкл Р03.01/02 / 1 = норма / 0 = авария *)
(* э.к.манометр Р03.01/01 / 1 = норма / 0 = нет давления *)
(* э.к.манометр Р03.01/02 / 1 = норма / 0 = нет давления *)
(* сигнал на пуск Р03.01/02 *)
(* авария Р03.01/02 *)
(* время задержки начала контроля параметра (например, задержка / контроля эк.манометра после насоса, время на разгон). *)
(* - низкий уровень в емкости V02.07 / (сигнал из АСУ-2 осмос 1) 1 = true *)
(* - высокий уровень в емкости V06.01 / (сигнал из АСУ-1 общий) 1 = true *)
(* - высокий уровень в емкости V04.01 / (сигнал от БМТ, МЕ04) 1 = true *)
(* Время задержки повторного пуска насосов, сек *)
(* авт.выкл и сигнал от самого доз.насоса Р03.02/02 / 1 = норма, 0 = авария *)
(* авт.выкл и сигнал от самого доз.насоса Р03.02/01 / 1 = норма, 0 = авария *)
(* Доз.насосы Р03.02/01 и Р03.02/02 на входе в осмос 2 *)
(* выход на пуск Р03.02/01 *)
(* задание производительности Р03.02/01 *)
(* задание производительности Р03.02/02 *)
(* выход на пуск Р03.02/02 *)
(* авария основного осмоса из / блока управления пусками *)
(* авария резервного осмоса из / блока управлени пусками *)
(* пуск основного осмоса *)
(* задержка контроля датчика РТ0301 *)
(* клапан 12 *)
(* клапан 14 *)
(* клапан 13 *)
(* клапан 18 *)
(* *авария основного осмоса по макс давлению датчика РТ03.03/01 *)
(* *авария основного осмоса по макс давлению датчика РТ03.04/01 *)
(* задержка до начала закрытия клапанов после выключения насоса *)
(* активен насос Р03.01/02 *)
(* активен насос Р03.01/01 *)
(* старт НД03.04/02 *)
(* пуск резервного осмоса *)
(* клапан 15 *)
(* клапан 17 *)
(* клапан 16 *)
(* *авария резервного осмоса по макс давлению датчика РТ03.03/01 *)
(* *авария резервного осмоса по макс давлению датчика РТ03.04/01 *)
#0 lowLevelV0207 <= boolStub
#1 AND(NOT lowLevelV0207, NOT highLevelV0601, NOT highLevelV0401)
#2 AND(NOT alarmP0302, NOT DD1_DI_13, NOT osmosTotalAlarm)
#3 AND(#1, #2)
#4 P0301:RichTwoPumpManager(#3, setWordP0301.0, setWordP0301.1, setWordP0301.2, setWordP0301.3, setWordP0301.4, setWordP0301.5, setWordP0301.6, setWordP0301.7, setWordP0301.8, setWordP0301.9, setWordP0301.10, resetAlarms, DELAY_REPEATED_START_SEC, setWordP0301.11, setWordP0301.12)
#5 statWordP0301.0 <= #4.out 1
#6 statWordP0301.1 <= #4.out 2
#7 statWordP0301.2 <= #4.out 3
#8 statWordP0301.3 <= #4.out 4
#9 counterP030101 <= #4.out 5
#10 counterP030102 <= #4.out 6
#11 daysOfWorkP030101 <= #4.out 7
#12 hoursOfWorkP030101 <= #4.out 8
#13 minutesOfWorkP030101 <= #4.out 9
#14 secondsOfWorkP030101 <= #4.out 10
#15 daysOfWorkP030102 <= #4.out 11
#16 hoursOfWorkP030102 <= #4.out 12
#17 minutesOfWorkP030102 <= #4.out 13
#18 secondsOfWorkP030102 <= #4.out 14
#19 statWordP0301.4 <= #4.out 15
#20 statWordP0301.5 <= #4.out 16
#21 toNextStarnP030101timer <= #4.out 17
#22 toNextStarnP030102timer <= #4.out 18
#23 statWordP0301.6 <= #4.out 19
#24 statWordP0301.7 <= #4.out 20
#25 delayCheckIfP030101works:TON(IN: #4.out 15, PT: CHECKING_DELAY_TIME)
#26 AND(NOT DD1_DI_3, #25.Q)
#27 OR(NOT DD1_DI_1, #26, lowPT030101_P030101, lowPT030102_P030101)
#28 setWordP0301.11 <= #27
#29 delayCheckIfP030102works:TON(IN: #4.out 16, PT: CHECKING_DELAY_TIME)
#30 AND(NOT DD1_DI_4, #29.Q)
#31 OR(NOT DD1_DI_2, #30, lowPT030101_P030102, lowPT030102_P030102)
#32 setWordP0301.12 <= #31
#33 highLevelV0601 <= boolStub
#34 highLevelV0401 <= boolStub
#35 CHECKING_DELAY_TIME <= T#5s
#36 DELAY_REPEATED_START_SEC <= 300
#37 DELAY_TO_OFF_VALVE <= T#3s
#38 DELAY_TO_CHECK_PT0301 <= T#10s
#39 MOVE(EN: testBool1, testReal1)
#40 testReal <= #39
#41 DELAY_TO_SWITCH_VALVE <= T#15s
#42 MOVE(EN: testBool2, testReal2)
#43 testReal <= #42
#44 DELAY_TO_CLOSE_VALVE <= T#10s
#45 testBlink:BLINK(ENABLE: TRUE, TIMELOW: T#500ms, TIMEHIGH: T#500ms)
#46 testBlinkIndikator <= #45.OUT
#47 MACRO обмен сигналами с DD2 (ПР102)()
	(* передача производительности / Р03.06/02 через модбас *)
	(* производительность доз.насоса Р03.06/02 / в процентах 0...100% *)
	(* 5430 - это число, соответствующее 100% / производительности ЧРП (50Гц) / так показали эксперименты в Казани / по РЭ и обучающим видео Овна 50Гц / соответствует число 16384 / Не знаю кому верить / Это число надо уточнить при ПНР... *)
	(* передача производительности / Р03.06/01 через модбас *)
	(* производительность доз.насоса Р03.06/01 / в процентах 0...100% *)
	(* сигнал на запуск Р03.06/02 *)
	(* получить из DD2 *)
	(* авария насоса Р03.06/02 *)
	(* передать в DD2 *)
	(* сигнал на запуск Р03.06/01 *)
	(* авария насоса Р03.06/01 *)
	(* есть авария хотя бы одного датчика в резеврном осмосе / получить из DD2 (ПР102), 1=авария *)
	(* сигнал на старт Р03.01/02 *)
	(* сигнал на старт Р03.01/01 *)
	#48 DO_bit_mask_DD2.0 <= statWordP0301.4
	#49 P030601alarm <= stat_word_P030601_PLC.3
	#50 DO_bit_mask_DD2.1 <= statWordP0301.5
	#51 P030602alarm <= stat_word_P030602_PLC.3
	#52 MACRO командное слово Р03.06/01(pin 1 "пуск/стоп": P030601start)
		(* не используется *)
		(* 0=набор 1, 1=набор 2 *)
		(* не используется *)
		(* 0=реле 1 выключено, 1=реле 1 включено *)
		(* 0=данные недействительны, 1=данные действительны *)
		(* 0=изменение скорости1 (согласно 3-4), 1=изменение скорости 2 (согласно 3-5) *)
		(* 0=работа по заданию, 1=фиксированная частота(параметр 3-11) *)
		(* 0=нет сброса, 1=сброс *)
		(* 0=останов с замедлением, 1=пуск *)
		(* фиксация частоты, 0=есть, 1=нет *)
		(* быстрый останов, 0=есть, 1=нет *)
		(* останов выбегом, 0=есть, 1=нет *)
		(* торможение постоянным током, 0=есть, 1=нет. *)
		(* предустановленное значение, старший бит, 0=0, 1=1 *)
		(* предустановленное значение, младший бит, 0=0, 1=1 *)
		#53 com_word_P030601_PLC.0 <= 0
		#54 com_word_P030601_PLC.1 <= 0
		#55 com_word_P030601_PLC.2 <= 1
		#56 com_word_P030601_PLC.3 <= pin 1
		#57 com_word_P030601_PLC.6 <= pin 1
		#58 com_word_P030601_PLC.4 <= 1
		#59 com_word_P030601_PLC.5 <= 1
		#60 com_word_P030601_PLC.7 <= 0
		#61 com_word_P030601_PLC.8 <= 0
		#62 com_word_P030601_PLC.9 <= 0
		#63 com_word_P030601_PLC.10 <= 1
		#64 com_word_P030601_PLC.11 <= 0
		#65 com_word_P030601_PLC.12 <= 0
		#66 com_word_P030601_PLC.13 <= 0
		#67 com_word_P030601_PLC.14 <= 0
	END_MACRO
	#68 MACRO командное слово Р03.06/02(pin 1 "пуск/стоп": P030602start)
		(* не используется *)
		(* 0=набор 1, 1=набор 2 *)
		(* не используется *)
		(* 0=реле 1 выключено, 1=реле 1 включено *)
		(* 0=данные недействительны, 1=данные действительны *)
		(* 0=изменение скорости1 (согласно 3-4), 1=изменение скорости 2 (согласно 3-5) *)
		(* 0=работа по заданию, 1=фиксированная частота(параметр 3-11) *)
		(* 0=нет сброса, 1=сброс *)
		(* 0=останов с замедлением, 1=пуск *)
		(* фиксация частоты, 0=есть, 1=нет *)
		(* быстрый останов, 0=есть, 1=нет *)
		(* останов выбегом, 0=есть, 1=нет *)
		(* торможение постоянным током, 0=есть, 1=нет. *)
		(* предустановленное значение, старший бит, 0=0, 1=1 *)
		(* предустановленное значение, младший бит, 0=0, 1=1 *)
		#69 com_word_P030602_PLC.0 <= 0
		#70 com_word_P030602_PLC.1 <= 0
		#71 com_word_P030602_PLC.2 <= 1
		#72 com_word_P030602_PLC.3 <= pin 1
		#73 com_word_P030602_PLC.6 <= pin 1
		#74 com_word_P030602_PLC.4 <= 1
		#75 com_word_P030602_PLC.5 <= 1
		#76 com_word_P030602_PLC.7 <= 0
		#77 com_word_P030602_PLC.8 <= 0
		#78 com_word_P030602_PLC.9 <= 0
		#79 com_word_P030602_PLC.10 <= 1
		#80 com_word_P030602_PLC.11 <= 0
		#81 com_word_P030602_PLC.12 <= 0
		#82 com_word_P030602_PLC.13 <= 0
		#83 com_word_P030602_PLC.14 <= 0
	END_MACRO
	#84 WORD_TO_BOOL(DI_bit_mask_DD2)
	#85 osmos2sensorsAlarm <= #84
	#86 freqP030601:LIN_TRAFO(IN: Yout_Total_P030601, IN_MIN: 0, IN_MAX: 100, OUT_MIN: 0, OUT_MAX: 16384)
	#87 REAL_TO_WORD(#86.OUT)
	#88 set_freq_P030601_PLC <= #87
	#89 MACRO обработка аналоговых сигналов датчиков резервного осмоса()
		(* Показания расходомера FIT03.01/01 на входе в осмос 2. / Для управления производительностью НД Р03.02 (1 и 2). *)
		(* давление датчик РТ03.01/02 *)
		(* давление датчик РТ03.02/02 *)
		(* давление датчик РТ03.03/02 *)
		(* давление датчик РТ03.04/02 *)
		(* расходомер FIT03.03/02 *)
		(* расходомер FIT03.02/02 *)
		(* кондуктомер QIT03.01/02 *)
		#90 pt030102:ControlAI(PT030102rawValue, -, PT030102maxValue)
		#91 PT030102realValue <= #90.out 1
		#92 PT030102alarm <= #90.out 2
		#93 pt030202:ControlAI(PT030202rawValue, -, PT030202maxValue)
		#94 PT030202realValue <= #93.out 1
		#95 PT030202alarm <= #93.out 2
		#96 pt030302:ControlAI(PT030302rawValue, -, PT030302maxValue)
		#97 PT030302realValue <= #96.out 1
		#98 PT030302alarm <= #96.out 2
		#99 pt030402:ControlAI(PT030402rawValue, -, PT030402maxValue)
		#100 PT030402realValue <= #99.out 1
		#101 PT030402alarm <= #99.out 2
		#102 fit0301:ControlAI(FIT030101rawValue, -, FIT0301maxValue)
		#103 flowFIT0301 <= #102.out 1
		#104 FIT0301alarm <= #102.out 2
		#105 fit030202:ControlAI(FIT030202rawValue, -, FIT030202maxValue)
		#106 FIT030202realValue <= #105.out 1
		#107 FIT030202alarm <= #105.out 2
		#108 fit030302:ControlAI(FIT030302rawValue, -, FIT030302maxValue)
		#109 FIT030302realValue <= #108.out 1
		#110 FIT030302alarm <= #108.out 2
		#111 qit030102:ControlAI(QIT030102rawValue, -, QIT030102maxValue)
		#112 QIT030102realValue <= #111.out 1
		#113 QIT030102alarm <= #111.out 2
	END_MACRO
	#114 freqP030602:LIN_TRAFO(IN: Yout_Total_P030602, IN_MIN: 0, IN_MAX: 100, OUT_MIN: 0, OUT_MAX: 16384)
	#115 REAL_TO_WORD(#114.OUT)
	#116 set_freq_P030602_PLC <= #115
END_MACRO
#117 MACRO обработка аналоговых сигналов датчиков основного осмоса()
	#118 controlAIpt030101:ControlAI(DD1_AI_2, -, PT030101maxValue)
	#119 PT030101realValue <= #118.out 1
	#120 PT030101alarm <= #118.out 2
	#121 controlAIpt030201:ControlAI(DD1_AI_3, -, PT030201maxValue)
	#122 PT030201realValue <= #121.out 1
	#123 PT030201alarm <= #121.out 2
	#124 controlAIpt030301:ControlAI(DD1_AI_4, -, PT030301maxValue)
	#125 PT030301realValue <= #124.out 1
	#126 PT030301alarm <= #124.out 2
	#127 controlAIpt030401:ControlAI(DD1_AI_5, -, PT030401maxValue)
	#128 PT030401realValue <= #127.out 1
	#129 PT030401alarm <= #127.out 2
	#130 controlAIqit030101:ControlAI(DD1_AI_6, -, QIT030101maxValue)
	#131 QIT030101realValue <= #130.out 1
	#132 QIT030101alarm <= #130.out 2
	#133 controlAIfit030201:ControlAI(DD1_AI_7, -, FIT030201maxValue)
	#134 FIT030201realValue <= #133.out 1
	#135 FIT030201alarm <= #133.out 2
	#136 controlAIfit030301:ControlAI(DD1_AI_8, -, FIT030301maxValue)
	#137 FIT030301realValue <= #136.out 1
	#138 FIT030301alarm <= #136.out 2
END_MACRO
#139 P0302:RichTwoPumpManager(startP0302, setWordP0302.0, setWordP0302.1, setWordP0302.2, setWordP0302.3, setWordP0302.4, setWordP0302.5, setWordP0302.6, setWordP0302.7, setWordP0302.8, setWordP0302.9, setWordP0302.10, resetAlarms, DELAY_REPEATED_START_SEC, setWordP0302.11, setWordP0302.12)
#140 statWordP0302.0 <= #139.out 1
#141 statWordP0302.1 <= #139.out 2
#142 statWordP0302.2 <= #139.out 3
#143 statWordP0302.3 <= #139.out 4
#144 counterP030201 <= #139.out 5
#145 counterP030202 <= #139.out 6
#146 daysOfWorkP030201 <= #139.out 7
#147 hoursOfWorkP030201 <= #139.out 8
#148 minutesOfWorkP030201 <= #139.out 9
#149 secondsOfWorkP030201 <= #139.out 10
#150 daysOfWorkP030202 <= #139.out 11
#151 hoursOfWorkP030202 <= #139.out 12
#152 minutesOfWorkP030202 <= #139.out 13
#153 secondsOfWorkP030202 <= #139.out 14
#154 statWordP0302.4 <= #139.out 15
#155 DD1_DO_2 <= #139.out 15
#156 DD1_DO_3 <= #139.out 16
#157 toNextStarnP030201timer <= #139.out 17
#158 statWordP0302.5 <= #139.out 16
#159 toNextStarnP030202timer <= #139.out 18
#160 statWordP0302.6 <= #139.out 19
#161 statWordP0302.7 <= #139.out 20
#162 OR(DD1_DI_11, DD1_DI_7, PT030101alarm, PT030201alarm, PT030301alarm, PT030401alarm, QIT030101alarm, FIT030201alarm, FIT030301alarm, P030601alarm)
#163 osmos1EquipmentAlarm <= #162
#164 OR(#162, statWordOsmos.6)
#165 OR(DD1_DI_12, DD1_DI_8, osmos2sensorsAlarm, P030602alarm)
#166 osmos2EquipmentAlarm <= #165
#167 OR(statWordOsmos.7, #165)
#168 AND(#164, #167)
#169 osmosTotalAlarm <= #168
#170 setWordP0302.11 <= NOT DD1_DI_5
#171 setWordP0302.12 <= NOT DD1_DI_6
#172 P0302dos:DosingPumpProportional(flowFIT0301, -, setMaxPumpDosingValueP0302, -, -, setKoeffProportionalityP0302, -)
#173 dosingErrorP0302 <= #172.out 2
#174 SEL(statWordP0302.4, 4.00, #172.out 1)
#175 DD1_AO_1 <= #174
#176 SEL(statWordP0302.5, 4.00, #172.out 1)
#177 DD1_AO_2 <= #176
#178 OR(statWordP0301.4, statWordP0301.5)
#179 OR(setWordOsmos.11, osmos1EquipmentAlarm, osmos1AlarmPT030301, osmos1AlarmPT030401)
#180 OR(setWordOsmos.12, osmos2EquipmentAlarm, osmos2AlarmPT030302, osmos2AlarmPT030402)
#181 osmosManager:RichTwoPumpManager(#178, setWordOsmos.0, setWordOsmos.1, setWordOsmos.2, setWordOsmos.3, setWordOsmos.4, setWordOsmos.5, setWordOsmos.6, setWordOsmos.7, setWordOsmos.8, setWordOsmos.9, setWordOsmos.10, resetAlarms, DELAY_REPEATED_START_SEC, #179, #180)
#182 statWordOsmos.0 <= #181.out 1
#183 statWordOsmos.1 <= #181.out 2
#184 statWordOsmos.2 <= #181.out 3
#185 statWordOsmos.3 <= #181.out 4
#186 counterOsmos1 <= #181.out 5
#187 counterOsmos2 <= #181.out 6
#188 daysOfWorkOsmos1 <= #181.out 7
#189 hoursOfWorkOsmos1 <= #181.out 8
#190 minutesOfWorkOsmos1 <= #181.out 9
#191 secondsOfWorkOsmos1 <= #181.out 10
#192 daysOfWorkOsmos2 <= #181.out 11
#193 hoursOfWorkOsmos2 <= #181.out 12
#194 minutesOfWorkOsmos2 <= #181.out 13
#195 secondsOfWorkOsmos2 <= #181.out 14
#196 statWordOsmos.4 <= #181.out 15
#197 statWordOsmos.5 <= #181.out 16
#198 toNextStarnOsmos1timer <= #181.out 17
#199 toNextStarnOsmos2timer <= #181.out 18
#200 statWordOsmos.6 <= #181.out 19
#201 statWordOsmos.7 <= #181.out 20
#202 MACRO основной осмос(pin 1 "пуск основного осмоса": statWordOsmos.4, pin 2 "текущие показания датчика РТ03.01/01, МПа": PT030101realValue, pin 3 "уставка датчиков РТ03.01 для старта, МПа": PT0301startValue, pin 4 "активен насос Р03.01/01": statWordP0301.4, pin 5 "активен насос Р03.01/02": statWordP0301.5, pin 6 "текущий расход FIT03,03/01, куб.м/час": FIT030301realValue, pin 7 "заданный расход FIT03,03/01, куб.м/час": FIT0303setValue, pin 8 "КР, расход осн.осм.": KP_F_P030601, pin 9 "I, расход осн.осм.": I_F_P030601, pin 10 "D, расход осн.осм.": D_F_P030601, pin 11 "текущее давление, РТ03.02/01, МПа": PT030201realValue, pin 12 "максимальное давление, РТ03.02/01, МПа": PT0302setMaxValue, pin 13 "КР, давление осн.осм.": KP_P_P030601, pin 14 "I, давление осн.осм.": I_P_P030601, pin 15 "D, давление осн.осм.": D_P_P030601, pin 16 "текущие показания датчика РТ03.03/01, МПа": PT030301realValue, pin 17 "уставка max давление РТ03.03, МПа": PT0303setMaxValue, pin 18 "текущие показания датчика РТ03.04/01, МПа": PT030401realValue, pin 19 "уставка max давление РТ03.04, МПа": PT0304setMaxValue)
	#203 MACRO 1 этап основной осмос(pin 1 "пуск основного осмоса": pin 1)
		#204 OR(pin 1, #211.Q)
		out 2 "клапан 12" <= #204
		#205 tonValve14:TON(IN: pin 1, PT: DELAY_TO_OFF_VALVE)
		#206 OR(#205.Q, #210.Q)
		out 1 "клапан 14/13" <= #206
		out 3 "старт НД03.04/01" <= #207.Q
		out 5 "startP0302" <= #207.Q
		#207 tonValve18:TON(IN: #205.Q, PT: DELAY_TO_OFF_VALVE)
		#208 OR(#207.Q, #209.Q)
		out 4 "клапан 18" <= #208
		#209 tofValve18:TOF(IN: #207.Q, PT: DELAY_TO_CLOSE_VALVE)
		#210 tofValve14:TOF(IN: #209.Q, PT: DELAY_TO_OFF_VALVE)
		#211 tofValve12:TOF(IN: #210.Q, PT: DELAY_TO_OFF_VALVE)
	END_MACRO
	out 7 "клапан 12" <= #203.out 2
	out 11 "старт НД03.04/01" <= #203.out 3
	out 10 "клапан 18" <= #203.out 4
	out 12 "старт доз.насосов Р03.02" <= #203.out 5
	#212 MACRO 2 этап основной осмос(pin 1 "управлять клапанами 13/14": #203.out 1, pin 2 "начать второй этап": #203.out 5, pin 3 "текущие показания датчика РТ03.01/01": pin 2, pin 4 "уставка датчиков РТ03.01 для старта": pin 3, pin 5 "активен насос Р03.01/01": pin 4, pin 6 "активен насос Р03.01/02": pin 5)
		#213 +(DELAY_TO_SWITCH_VALVE, DELAY_TO_CLOSE_VALVE)
		#214 tonSwitchValve1413:TON(IN: #218, PT: DELAY_TO_SWITCH_VALVE)
		#215 HoldingToEndProcValve:TOF(IN: #214.Q, PT: #213)
		#216 SEL(#215.Q, pin 1, #220.Q)
		out 1 "клапан 14" <= #216
		#217 >(pin 3, pin 4)
		#218 AND(#217, #221.Q)
		out 5 "пуск насоса Р03.06/01" <= #218
		#219 valve1413switcher:IfBOOL(key: #215.Q, input: pin 1)
		#220 delayToSwitchValve14to13:TOF(IN: #219.keyFALSE, PT: DELAY_TO_OFF_VALVE)
		out 2 "клапан 13" <= #219.keyTRUE
		#221 tonPT030101:TON(IN: pin 2, PT: DELAY_TO_CHECK_PT0301)
		#222 AND(pin 5, #223)
		out 3 "авария насоса Р03.01/01" <= #222
		#223 AND(#221.Q, #224)
		#224 <(pin 3, pin 4)
		#225 AND(#223, pin 6)
		out 4 "авария насоса Р03.01/ 02" <= #225
	END_MACRO
	out 9 "клапан 14" <= #212.out 1
	out 8 "клапан 13" <= #212.out 2
	out 13 "авария низкое давление насос Р03.01/01" <= #212.out 3
	out 14 "авария низкое давление насос Р03.01/02" <= #212.out 4
	out 1 "пуск насоса Р03.06/01" <= #212.out 5
	#226 AND(#212.out 5, #227)
	out 2 "авария осмос 1  макс.давл.РТ03.03/01" <= #226
	#227 >=(pin 16, pin 17)
	#228 AND(#212.out 5, #229)
	out 3 "авария осмос 1  макс.давл.РТ03.04/01" <= #228
	#229 >=(pin 18, pin 19)
	#230 MACRO управление производительностью Р03.06/01(pin 1 "текущий расход, FIT03.03/01, куб.м/час": pin 6, pin 2 "заданный расход, FIT03.03/01 , куб.м/час": pin 7, pin 3 "КР, расход": pin 8, pin 4 "I, сек, расход": pin 9, pin 5 "D, сек, расход": pin 10, pin 6 "текущее давление, РТ03.02/01, МПа": pin 11, pin 7 "максимальное давление, РТ03.02/01, МПа": pin 12, pin 8 "КР, давление": pin 13, pin 9 "I, сек, давление": pin 14, pin 10 "D, сек, давление": pin 15)
		(* Задача: поддерживать заданный расход. / Если давление при этом превысит заданный уровень, / снижать производительность, не глядя на расход. / В идеале два ПИД-регулятора ПЛАВНО передают управление друг-другу. / Если реальность оказалась более сурова и регуляторы мешают друг другу, / то есть два пути: / 1. Настраивать ПИД-регуляторы коэффициентами / 2. Переосмысливать и переделывать этот блок. *)
		(* tесли выход менььше нуля, то ноль, / иначе - то, что насчитали *)
		#231 F_P030601:PID(ACTUAL: pin 1, SET_POINT: pin 2, KP: pin 3, TN: pin 4, TV: pin 5, Y_MANUAL: -, Y_OFFSET: -, Y_MIN: 0, Y_MAX: 100, MANUAL: -, RESET: #231.OVERFLOW)
		out 1 "производительность по расходу, 0...100%" <= #231.Y
		#232 <(#234, 0)
		#233 SEL(#232, #234, 0)
		out 3 "производительность итог, 0...100%" <= #233
		#234 -(#231.Y, #235)
		#235 -(100, #236.Y)
		out 2 "коррекция по давлению, 0...100%" <= #235
		#236 P_P030601:PID(ACTUAL: pin 6, SET_POINT: pin 7, KP: pin 8, TN: pin 9, TV: pin 10, Y_MANUAL: -, Y_OFFSET: -, Y_MIN: 0, Y_MAX: 100, MANUAL: -, RESET: #236.OVERFLOW)
	END_MACRO
	out 4 "производительность по расходу осн.осмос, 0...100%" <= #230.out 1
	out 5 "коррекция по давлению осн.осмос, 0...100%" <= #230.out 2
	out 6 "производительность итог осн.осмос, 0...100%" <= #230.out 3
END_MACRO
#237 P030601start <= #202.out 1
#238 osmos1AlarmPT030301 <= #202.out 2
#239 osmos1AlarmPT030401 <= #202.out 3
#240 Yout_F_P030601 <= #202.out 4
#241 Yout_P_P030601 <= #202.out 5
#242 Yout_Total_P030601 <= #202.out 6
#243 DD1_DO_6 <= #202.out 7
#244 DD1_DO_7 <= #202.out 8
#245 DD1_DO_8 <= #202.out 9
#246 DD1_DO_4 <= #202.out 11
#247 lowPT030101_P030101 <= #202.out 13
#248 lowPT030101_P030102 <= #202.out 14
#249 MACRO резервный осмос(pin 1 "пуск резервного осмоса": statWordOsmos.5, pin 2 "текущие показания РТ01.03/02": PT030102realValue, pin 3 "уставка РТ03.01/02 для старта": PT0301startValue, pin 4 "активен насос Р03.01/01": statWordP0301.4, pin 5 "активен насос Р03.01/02": statWordP0301.5, pin 6 "текущий расход, FIT03/03/02, куб.м/час": FIT030302realValue, pin 7 "заданный расход, FIT03/03/02, куб.м/час": FIT0303setValue, pin 8 "KP, расход, осмос 2": KP_F_P030602, pin 9 "I, расход, осмос 2": I_F_P030602, pin 10 "D, расход, осмос 2": D_F_P030602, pin 11 "текущее давление PT03.02/02, МПа": PT030202realValue, pin 12 "максимальное давление PT03.02/02, МПа": PT0302setMaxValue, pin 13 "KP, давление, осмос 2": KP_P_P030602, pin 14 "I, давление, осмос 2": I_P_P030602, pin 15 "D, давление, осмос 2": D_P_P030602, pin 16 "текущее давление РТ03.03/02": PT030302realValue, pin 17 "задание max давление РТ03.03/02": PT0303setMaxValue, pin 18 "текущее давление РТ03.04/02": PT030402realValue, pin 19 "задание max давление РТ03.04/02": PT0304setMaxValue)
	#250 MACRO 1 этап резервный осмос(pin 1 "пуск резервного осмоса": pin 1)
		#251 OR(pin 1, #258.Q)
		out 2 "клапан 15" <= #251
		#252 tonValve17:TON(IN: pin 1, PT: DELAY_TO_OFF_VALVE)
		#253 OR(#252.Q, #257.Q)
		out 1 "клапан 16/17" <= #253
		out 3 "старт НД03.04/02" <= #254.Q
		out 5 "startP0302" <= #254.Q
		#254 tonValve18rez:TON(IN: #252.Q, PT: DELAY_TO_OFF_VALVE)
		#255 OR(#254.Q, #256.Q)
		out 4 "клапан 18" <= #255
		#256 tofValve18rez:TOF(IN: #254.Q, PT: DELAY_TO_CLOSE_VALVE)
		#257 tofValve17:TOF(IN: #256.Q, PT: DELAY_TO_OFF_VALVE)
		#258 tofValve15:TOF(IN: #257.Q, PT: DELAY_TO_OFF_VALVE)
	END_MACRO
	out 5 "клапан 15" <= #250.out 2
	out 6 "старт НД03.04/02" <= #250.out 3
	out 2 "клапан 18" <= #250.out 4
	out 1 "пуск Р0302" <= #250.out 5
	#259 MACRO 2 этап резервный осмос(pin 1 "управлять клапанами 16/17": #250.out 1, pin 2 "начать второй этап": #250.out 5, pin 3 "текущие показания датчика РТ03.01/02": pin 2, pin 4 "уставка датчиков РТ03.01 для старта": pin 3, pin 5 "активен насос Р03.01/01": pin 4, pin 6 "активен насос Р03.01/02": pin 5)
		#260 +(DELAY_TO_SWITCH_VALVE, DELAY_TO_CLOSE_VALVE)
		#261 tonSwitchValve1716:TON(IN: #265, PT: DELAY_TO_SWITCH_VALVE)
		#262 HoldingToEndProcValveRez:TOF(IN: #261.Q, PT: #260)
		#263 SEL(#262.Q, pin 1, #267.Q)
		out 1 "клапан 17" <= #263
		#264 >(pin 3, pin 4)
		#265 AND(#264, #268.Q)
		out 5 "пуск насоса Р03.06/02" <= #265
		#266 valve1716switcher:IfBOOL(key: #262.Q, input: pin 1)
		#267 delayToSwitchValve17to16:TOF(IN: #266.keyFALSE, PT: DELAY_TO_OFF_VALVE)
		out 2 "клапан 16" <= #266.keyTRUE
		#268 tonPT030102:TON(IN: pin 2, PT: DELAY_TO_CHECK_PT0301)
		#269 AND(pin 5, #270)
		out 3 "авария насоса Р03.01/01" <= #269
		#270 AND(#268.Q, #271)
		#271 <(pin 3, pin 4)
		#272 AND(#270, pin 6)
		out 4 "авария насоса Р03.01/ 02" <= #272
	END_MACRO
	out 3 "клапан 17" <= #259.out 1
	out 4 "клапан 16" <= #259.out 2
	out 7 "авария низкое давление насос Р03.03/01" <= #259.out 3
	out 8 "авария низкое давление насос Р03.03/02" <= #259.out 4
	out 9 "пуск насоса Р03.06/02" <= #259.out 5
	#273 AND(#259.out 5, #274)
	out 13 "авария осмос 2 max давление РТ03.03/02" <= #273
	#274 >=(pin 16, pin 17)
	#275 AND(#259.out 5, #276)
	out 14 "авария осмос 2 max давление РТ03.04/02" <= #275
	#276 >=(pin 18, pin 19)
	#277 MACRO управление производительностью Р03.06/02(pin 1 "текущий расход, FIT03.03/02, куб.м/час": pin 6, pin 2 "заданный расход, FIT03.03/02 , куб.м/час": pin 7, pin 3 "КР, расход, осмос 2": pin 8, pin 4 "I, сек, расход, осмос 2": pin 9, pin 5 "D, сек, расход, осмос 2": pin 10, pin 6 "текущее давление, РТ03.02/02, МПа": pin 11, pin 7 "максимальное давление, РТ03.02/02, МПа": pin 12, pin 8 "КР, давление, осмос 2": pin 13, pin 9 "I, сек, давление, осмос 2": pin 14, pin 10 "D, сек, давление, осмос 2": pin 15)
		(* Задача: поддерживать заданный расход. / Если давление при этом превысит заданный уровень, / снижать производительность, не глядя на расход. / В идеале два ПИД-регулятора ПЛАВНО передают управление друг-другу. / Если реальность оказалась более сурова и регуляторы мешают друг другу, / то есть два пути: / 1. Настраивать ПИД-регуляторы коэффициентами / 2. Переосмысливать и переделывать этот блок. *)
		(* tесли выход менььше нуля, то ноль, / иначе - то, что насчитали *)
		#278 F_P030602:PID(ACTUAL: pin 1, SET_POINT: pin 2, KP: pin 3, TN: pin 4, TV: pin 5, Y_MANUAL: -, Y_OFFSET: -, Y_MIN: 0, Y_MAX: 100, MANUAL: -, RESET: #278.OVERFLOW)
		out 1 "производительность по расходу, 0...100%" <= #278.Y
		#279 <(#281, 0)
		#280 SEL(#279, #281, 0)
		out 3 "производительность итог, 0...100%" <= #280
		#281 -(#278.Y, #282)
		#282 -(100, #283.Y)
		out 2 "коррекция по давлению, 0...100%" <= #282
		#283 P_P030602:PID(ACTUAL: pin 6, SET_POINT: pin 7, KP: pin 8, TN: pin 9, TV: pin 10, Y_MANUAL: -, Y_OFFSET: -, Y_MIN: 0, Y_MAX: 100, MANUAL: -, RESET: #283.OVERFLOW)
	END_MACRO
	out 10 "производительность по расходу, рез.осмос, 0...100%" <= #277.out 1
	out 11 "коррекция по давлению, рез.осмос, 0...100%" <= #277.out 2
	out 12 "производительность итог, 0...100%" <= #277.out 3
END_MACRO
#284 DD1_DO_11 <= #249.out 3
#285 DD1_DO_10 <= #249.out 4
#286 DD1_DO_9 <= #249.out 5
#287 DD1_DO_5 <= #249.out 6
#288 lowPT030102_P030101 <= #249.out 7
#289 lowPT030102_P030102 <= #249.out 8
#290 P030602start <= #249.out 9
#291 Yout_F_P030602 <= #249.out 10
#292 Yout_P_P030602 <= #249.out 11
#293 Yout_Total_P030602 <= #249.out 12
#294 osmos2AlarmPT030302 <= #249.out 13
#295 osmos2AlarmPT030402 <= #249.out 14
#296 OR(#202.out 10, #249.out 2)
#297 DD1_DO_1 <= #296
#298 OR(#202.out 12, #249.out 1)
#299 startP0302 <= #298
_END_CFC_
END_PROGRAM
